C08959=1014.660,111.071,-128.777,-24.334,21.425,-41.690
C08960=1014.666,110.672,-128.741,-24.334,21.425,-41.694
C08961=1014.672,110.274,-128.704,-24.333,21.425,-41.697
C08962=1014.678,109.875,-128.668,-24.333,21.425,-41.701
C08963=1014.685,109.477,-128.631,-24.332,21.426,-41.703
C08964=1014.691,109.078,-128.595,-24.332,21.426,-41.707
C08965=1014.697,108.680,-128.557,-24.331,21.426,-41.710
C08966=1014.703,108.282,-128.521,-24.331,21.426,-41.714
C08967=1014.710,107.883,-128.485,-24.330,21.426,-41.717
C08968=1014.715,107.485,-128.448,-24.330,21.427,-41.719
C08969=1014.722,107.086,-128.411,-24.330,21.427,-41.723
C08970=1014.728,106.687,-128.374,-24.329,21.427,-41.727
C08971=1014.734,106.289,-128.338,-24.328,21.427,-41.730
C08972=1014.740,105.890,-128.301,-24.328,21.428,-41.734
C08973=1014.746,105.492,-128.265,-24.328,21.428,-41.736
C08974=1014.752,105.093,-128.228,-24.327,21.429,-41.740
C08975=1014.758,104.695,-128.192,-24.327,21.429,-41.743
C08976=1014.763,104.296,-128.155,-24.326,21.429,-41.747
C08977=1014.770,103.898,-128.118,-24.326,21.429,-41.751
C08978=1014.776,103.499,-128.082,-24.325,21.430,-41.754
C08979=1014.781,103.100,-128.044,-24.325,21.430,-41.756
C08980=1014.787,102.702,-128.008,-24.324,21.430,-41.760
C08981=1014.793,102.303,-127.972,-24.324,21.430,-41.763
C08982=1014.799,101.904,-127.935,-24.323,21.430,-41.767
C08983=1014.805,101.506,-127.898,-24.323,21.431,-41.771
C08984=1014.810,101.107,-127.862,-24.322,21.431,-41.775
C08985=1014.816,100.708,-127.826,-24.322,21.431,-41.778
C08986=1014.821,100.309,-127.789,-24.322,21.432,-41.780
C08987=1014.827,99.912,-127.752,-24.321,21.432,-41.784
C08988=1014.833,99.513,-127.716,-24.320,21.432,-41.787
C08989=1014.839,99.114,-127.679,-24.320,21.432,-41.791
C08990=1014.844,98.715,-127.643,-24.319,21.433,-41.795
C08991=1014.849,98.316,-127.606,-24.319,21.432,-41.798
C08992=1014.855,97.917,-127.569,-24.318,21.433,-41.802
C08993=1014.861,97.518,-127.533,-24.318,21.433,-41.806
C08994=1014.866,97.120,-127.497,-24.318,21.434,-41.808
C08995=1014.871,96.721,-127.459,-24.317,21.434,-41.811
C08996=1014.877,96.322,-127.423,-24.317,21.435,-41.815
C08997=1014.883,95.923,-127.386,-24.316,21.435,-41.819
C08998=1014.888,95.524,-127.350,-24.316,21.435,-41.822
C08999=1014.893,95.125,-127.314,-24.315,21.435,-41.826
C09000=1014.898,94.727,-127.277,-24.315,21.436,-41.830
C09001=1014.904,94.328,-127.240,-24.314,21.435,-41.833
C09002=1014.910,93.929,-127.204,-24.313,21.436,-41.837
C09003=1014.915,93.530,-127.168,-24.313,21.436,-41.841
C09004=1014.920,93.131,-127.131,-24.312,21.437,-41.844
C09005=1014.925,92.732,-127.095,-24.312,21.437,-41.846
C09006=1014.930,92.333,-127.057,-24.312,21.437,-41.850
C09007=1014.936,91.934,-127.021,-24.311,21.438,-41.854
C09008=1014.940,91.535,-126.985,-24.311,21.438,-41.857
C09009=1014.946,91.136,-126.948,-24.310,21.438,-41.861
C09010=1014.951,90.737,-126.912,-24.310,21.438,-41.865
C09011=1014.956,90.337,-126.875,-24.309,21.439,-41.868
C09012=1014.961,89.938,-126.839,-24.309,21.439,-41.872
C09013=1014.966,89.540,-126.802,-24.308,21.439,-41.875
C09014=1014.971,89.148,-126.766,-24.308,21.439,-41.879
C09015=1014.976,88.761,-126.731,-24.307,21.440,-41.883
C09016=1014.981,88.378,-126.696,-24.307,21.440,-41.887
C09017=1014.985,87.995,-126.662,-24.306,21.440,-41.890
C09018=1014.991,87.607,-126.625,-24.305,21.440,-41.894
C09019=1014.996,87.211,-126.590,-24.305,21.441,-41.898
C09020=1015.001,86.807,-126.553,-24.304,21.441,-41.901
C09021=1015.005,86.403,-126.516,-24.304,21.442,-41.905
C09022=1015.010,85.994,-126.479,-24.303,21.441,-41.908
C09023=1015.016,85.586,-126.441,-24.303,21.442,-41.912
C09024=1015.020,85.175,-126.405,-24.302,21.442,-41.916
C09025=1015.025,84.763,-126.366,-24.302,21.443,-41.920
C09026=1015.031,84.349,-126.328,-24.301,21.443,-41.923
C09027=1015.035,83.933,-126.291,-24.301,21.443,-41.927
C09028=1015.040,83.516,-126.253,-24.300,21.444,-41.931
C09029=1015.046,83.097,-126.214,-24.300,21.444,-41.935
C09030=1015.050,82.677,-126.176,-24.299,21.444,-41.938
C09031=1015.055,82.256,-126.138,-24.299,21.444,-41.942
C09032=1015.057,82.045,-126.118,-24.299,21.445,-41.944
C09033=1015.060,81.833,-126.099,-24.298,21.444,-41.947
C09034=1015.062,81.621,-126.080,-24.298,21.445,-41.949
C09035=1015.065,81.409,-126.061,-24.298,21.445,-41.951
C09036=1015.067,81.197,-126.041,-24.297,21.445,-41.953
C09037=1015.069,80.985,-126.022,-24.297,21.445,-41.955
C09038=1015.072,80.772,-126.002,-24.297,21.445,-41.956
C09039=1015.074,80.559,-125.983,-24.297,21.446,-41.958
C09040=1015.077,80.346,-125.963,-24.296,21.446,-41.960
C09041=1015.079,80.133,-125.945,-24.296,21.446,-41.962
C09042=1015.081,79.922,-125.925,-24.296,21.446,-41.964
C09043=1015.084,79.712,-125.906,-24.296,21.447,-41.966
C09044=1015.089,79.298,-125.869,-24.295,21.447,-41.970
C09045=1015.093,78.892,-125.831,-24.294,21.447,-41.973
C09046=1015.098,78.495,-125.795,-24.294,21.447,-41.977
C09047=1015.103,78.104,-125.760,-24.293,21.448,-41.980
C09048=1015.107,77.717,-125.725,-24.293,21.447,-41.986
C09049=1015.110,77.332,-125.690,-24.292,21.448,-41.989
C09050=1015.114,76.943,-125.655,-24.292,21.449,-41.994
C09051=1015.119,76.549,-125.619,-24.291,21.449,-41.997
C09052=1015.123,76.147,-125.582,-24.291,21.449,-42.001
C09053=1015.128,75.735,-125.545,-24.290,21.450,-42.004
C09054=1015.132,75.316,-125.507,-24.290,21.450,-42.008
C09055=1015.134,75.103,-125.487,-24.289,21.451,-42.010
C09056=1015.137,74.889,-125.468,-24.289,21.451,-42.012
C09057=1015.140,74.676,-125.449,-24.289,21.450,-42.015
C09058=1015.141,74.462,-125.430,-24.288,21.451,-42.017
C09059=1015.143,74.249,-125.409,-24.288,21.451,-42.019
C09060=1015.146,74.036,-125.391,-24.288,21.451,-42.021
C09061=1015.148,73.825,-125.372,-24.288,21.451,-42.023
C09062=1015.151,73.614,-125.352,-24.287,21.452,-42.025
C09063=1015.154,73.193,-125.314,-24.287,21.452,-42.028
C09064=1015.159,72.776,-125.276,-24.286,21.452,-42.034
C09065=1015.164,72.360,-125.239,-24.285,21.452,-42.037
C09066=1015.168,71.946,-125.201,-24.285,21.453,-42.041
C09067=1015.172,71.534,-125.164,-24.285,21.453,-42.045
C09068=1015.176,71.123,-125.127,-24.284,21.454,-42.049
C09069=1015.181,70.713,-125.090,-24.283,21.453,-42.054
C09070=1015.184,70.302,-125.052,-24.283,21.454,-42.058
C09071=1015.189,69.890,-125.015,-24.282,21.454,-42.061
C09072=1015.193,69.479,-124.978,-24.282,21.455,-42.065
C09073=1015.197,69.069,-124.941,-24.281,21.455,-42.069
C09074=1015.201,68.660,-124.904,-24.280,21.455,-42.074
C09075=1015.205,68.253,-124.867,-24.280,21.456,-42.078
C09076=1015.209,67.847,-124.830,-24.279,21.456,-42.082
C09077=1015.212,67.443,-124.794,-24.279,21.457,-42.085
C09078=1015.216,67.039,-124.757,-24.278,21.457,-42.089
C09079=1015.221,66.637,-124.721,-24.278,21.457,-42.094
C09080=1015.225,66.236,-124.685,-24.277,21.457,-42.098
C09081=1015.228,65.838,-124.649,-24.277,21.458,-42.102
C09082=1015.232,65.430,-124.612,-24.276,21.458,-42.106
C09083=1015.234,65.217,-124.593,-24.276,21.459,-42.108
C09084=1015.236,64.996,-124.574,-24.275,21.458,-42.111
C09085=1015.238,64.766,-124.553,-24.275,21.458,-42.113
C09086=1015.241,64.530,-124.531,-24.275,21.459,-42.115
C09087=1015.242,64.294,-124.510,-24.274,21.459,-42.116
C09088=1015.245,64.065,-124.489,-24.274,21.459,-42.120
C09089=1015.247,63.847,-124.470,-24.274,21.460,-42.122
C09090=1015.250,63.431,-124.432,-24.273,21.459,-42.127
C09091=1015.252,63.192,-124.410,-24.273,21.460,-42.129
C09092=1015.255,62.934,-124.387,-24.272,21.460,-42.131
C09093=1015.258,62.653,-124.362,-24.272,21.460,-42.133
C09094=1015.262,62.233,-124.324,-24.271,21.461,-42.139
C09095=1015.265,61.832,-124.289,-24.271,21.461,-42.142
C09096=1015.268,61.432,-124.252,-24.270,21.462,-42.146
C09097=1015.273,61.032,-124.217,-24.270,21.462,-42.150
C09098=1015.276,60.632,-124.181,-24.269,21.462,-42.155
C09099=1015.279,60.232,-124.145,-24.269,21.463,-42.159
C09100=1015.283,59.832,-124.109,-24.268,21.463,-42.163
C09101=1015.286,59.432,-124.072,-24.268,21.464,-42.166
C09102=1015.289,59.031,-124.037,-24.267,21.463,-42.172
C09103=1015.293,58.631,-124.000,-24.266,21.464,-42.175
C09104=1015.297,58.231,-123.965,-24.266,21.464,-42.179
C09105=1015.300,57.831,-123.929,-24.265,21.465,-42.183
C09106=1015.304,57.431,-123.894,-24.264,21.465,-42.188
C09107=1015.307,57.031,-123.858,-24.264,21.465,-42.192
C09108=1015.310,56.631,-123.822,-24.264,21.466,-42.196
C09109=1015.314,56.231,-123.785,-24.263,21.465,-42.201
C09110=1015.317,55.830,-123.750,-24.262,21.467,-42.205
C09111=1015.320,55.430,-123.714,-24.262,21.467,-42.209
C09112=1015.324,55.030,-123.679,-24.261,21.468,-42.212
C09113=1015.327,54.630,-123.642,-24.260,21.468,-42.218
C09114=1015.330,54.230,-123.607,-24.260,21.468,-42.221
C09115=1015.333,53.830,-123.571,-24.259,21.468,-42.225
C09116=1015.337,53.429,-123.536,-24.259,21.468,-42.230
C09117=1015.340,53.029,-123.499,-24.258,21.469,-42.234
C09118=1015.343,52.629,-123.464,-24.258,21.469,-42.238
C09119=1015.346,52.229,-123.428,-24.257,21.469,-42.243
C09120=1015.348,51.830,-123.392,-24.256,21.470,-42.247
C09121=1015.352,51.429,-123.357,-24.256,21.471,-42.251
C09122=1015.355,51.029,-123.321,-24.255,21.471,-42.255
C09123=1015.358,50.629,-123.285,-24.255,21.471,-42.260
C09124=1015.361,50.228,-123.249,-24.254,21.472,-42.264
C09125=1015.364,49.828,-123.214,-24.254,21.472,-42.268
C09126=1015.366,49.428,-123.178,-24.253,21.472,-42.273
C09127=1015.370,49.028,-123.143,-24.252,21.473,-42.277
C09128=1015.373,48.628,-123.106,-24.251,21.472,-42.282
C09129=1015.375,48.228,-123.072,-24.251,21.474,-42.286
C09130=1015.378,47.828,-123.036,-24.251,21.474,-42.290
C09131=1015.382,47.427,-123.000,-24.250,21.474,-42.295
C09132=1015.384,47.028,-122.965,-24.249,21.475,-42.299
C09133=1015.388,46.627,-122.929,-24.249,21.475,-42.302
C09134=1015.390,46.228,-122.894,-24.248,21.475,-42.308
C09135=1015.393,45.827,-122.858,-24.247,21.475,-42.311
C09136=1015.396,45.428,-122.823,-24.247,21.477,-42.316
C09137=1015.399,45.027,-122.787,-24.246,21.477,-42.321
C09138=1015.401,44.628,-122.752,-24.246,21.477,-42.325
C09139=1015.404,44.227,-122.716,-24.245,21.477,-42.330
C09140=1015.406,43.827,-122.681,-24.244,21.477,-42.333
C09141=1015.409,43.427,-122.646,-24.244,21.479,-42.338
C09142=1015.412,43.027,-122.610,-24.243,21.479,-42.343
C09143=1015.415,42.627,-122.575,-24.243,21.479,-42.347
C09144=1015.417,42.227,-122.539,-24.242,21.479,-42.352
C09145=1015.420,41.827,-122.504,-24.241,21.479,-42.356
C09146=1015.423,41.427,-122.468,-24.241,21.480,-42.359
C09147=1015.425,41.028,-122.433,-24.240,21.481,-42.365
C09148=1015.428,40.628,-122.398,-24.240,21.481,-42.369
C09149=1015.430,40.228,-122.362,-24.239,21.481,-42.374
C09150=1015.433,39.828,-122.327,-24.238,21.481,-42.378
C09151=1015.436,39.428,-122.292,-24.238,21.482,-42.383
C09152=1015.438,39.027,-122.256,-24.237,21.483,-42.387
C09153=1015.440,38.628,-122.221,-24.237,21.483,-42.391
C09154=1015.443,38.228,-122.186,-24.236,21.483,-42.396
C09155=1015.445,37.828,-122.151,-24.235,21.483,-42.400
C09156=1015.447,37.429,-122.115,-24.235,21.484,-42.405
C09157=1015.450,37.028,-122.080,-24.234,21.485,-42.409
C09158=1015.452,36.629,-122.045,-24.233,21.484,-42.414
C09159=1015.455,36.229,-122.010,-24.233,21.485,-42.418
C09160=1015.457,35.829,-121.974,-24.232,21.486,-42.424
C09161=1015.459,35.429,-121.940,-24.231,21.486,-42.428
C09162=1015.462,35.030,-121.905,-24.231,21.486,-42.433
C09163=1015.464,34.630,-121.869,-24.230,21.486,-42.437
C09164=1015.466,34.230,-121.834,-24.229,21.487,-42.442
C09165=1015.468,33.831,-121.799,-24.229,21.488,-42.446
C09166=1015.471,33.431,-121.764,-24.228,21.487,-42.451
C09167=1015.473,33.031,-121.729,-24.228,21.489,-42.455
C09168=1015.475,32.632,-121.694,-24.227,21.489,-42.461
C09169=1015.477,32.232,-121.659,-24.226,21.489,-42.464
C09170=1015.480,31.832,-121.624,-24.226,21.489,-42.469
C09171=1015.481,31.433,-121.589,-24.225,21.490,-42.474
C09172=1015.484,31.033,-121.554,-24.224,21.490,-42.479
C09173=1015.485,30.634,-121.519,-24.224,21.491,-42.483
C09174=1015.488,30.234,-121.484,-24.223,21.491,-42.488
C09175=1015.490,29.834,-121.449,-24.223,21.492,-42.492
C09176=1015.492,29.435,-121.414,-24.222,21.492,-42.497
C09177=1015.494,29.036,-121.379,-24.221,21.492,-42.501
C09178=1015.495,28.636,-121.345,-24.221,21.493,-42.507
C09179=1015.498,28.236,-121.309,-24.220,21.493,-42.510
C09180=1015.499,27.837,-121.274,-24.219,21.493,-42.516
C09181=1015.502,27.438,-121.240,-24.219,21.495,-42.520
C09182=1015.503,27.039,-121.205,-24.218,21.494,-42.525
C09183=1015.506,26.639,-121.170,-24.218,21.495,-42.529
C09184=1015.508,26.239,-121.136,-24.217,21.496,-42.534
C09185=1015.509,25.840,-121.101,-24.216,21.496,-42.540
C09186=1015.511,25.441,-121.066,-24.215,21.496,-42.543
C09187=1015.512,25.042,-121.031,-24.215,21.497,-42.549
C09188=1015.515,24.642,-120.997,-24.214,21.497,-42.553
C09189=1015.516,24.243,-120.962,-24.213,21.497,-42.558
C09190=1015.518,23.860,-120.929,-24.213,21.498,-42.562
C09191=1015.520,23.530,-120.899,-24.213,21.498,-42.564
C09192=1015.521,23.258,-120.876,-24.212,21.498,-42.567
C09193=1015.522,23.024,-120.856,-24.211,21.499,-42.573
C09194=1015.523,22.791,-120.836,-24.211,21.500,-42.577
C09195=1015.524,22.526,-120.812,-24.211,21.500,-42.580
C09196=1015.526,22.204,-120.785,-24.210,21.500,-42.584
C09197=1015.527,21.829,-120.752,-24.210,21.501,-42.586
C09198=1015.529,21.415,-120.717,-24.209,21.501,-42.593
C09199=1015.529,21.171,-120.695,-24.208,21.501,-42.597
C09200=1015.530,20.899,-120.671,-24.208,21.502,-42.599
C09201=1015.532,20.607,-120.647,-24.207,21.501,-42.602
C09202=1015.533,20.310,-120.621,-24.207,21.501,-42.604
C09203=1015.534,20.022,-120.596,-24.207,21.503,-42.606
C09204=1015.536,19.758,-120.573,-24.206,21.502,-42.610
C09205=1015.536,19.521,-120.552,-24.206,21.503,-42.613
C09206=1015.537,19.310,-120.535,-24.205,21.503,-42.617
C09207=1015.538,18.913,-120.500,-24.205,21.503,-42.622
C09208=1015.540,18.516,-120.466,-24.204,21.503,-42.626
C09209=1015.541,18.120,-120.431,-24.203,21.504,-42.632
C09210=1015.543,17.726,-120.398,-24.203,21.505,-42.635
C09211=1015.544,17.332,-120.363,-24.202,21.505,-42.641
C09212=1015.545,16.938,-120.330,-24.201,21.505,-42.646
C09213=1015.547,16.546,-120.296,-24.201,21.506,-42.650
C09214=1015.548,16.153,-120.262,-24.200,21.506,-42.656
C09215=1015.550,15.763,-120.228,-24.200,21.507,-42.659
C09216=1015.551,15.372,-120.195,-24.199,21.507,-42.665
C09217=1015.553,14.983,-120.161,-24.198,21.508,-42.670
C09218=1015.553,14.594,-120.128,-24.198,21.508,-42.674
C09219=1015.555,14.206,-120.094,-24.197,21.509,-42.680
C09220=1015.556,13.818,-120.061,-24.196,21.509,-42.683
C09221=1015.557,13.431,-120.028,-24.196,21.509,-42.689
C09222=1015.559,13.044,-119.994,-24.195,21.511,-42.693
C09223=1015.560,12.658,-119.961,-24.194,21.510,-42.698
C09224=1015.561,12.270,-119.929,-24.193,21.510,-42.703
C09225=1015.563,11.884,-119.895,-24.193,21.512,-42.707
C09226=1015.563,11.498,-119.862,-24.192,21.511,-42.713
C09227=1015.564,11.113,-119.829,-24.192,21.512,-42.716
C09228=1015.566,10.729,-119.796,-24.191,21.513,-42.722
C09229=1015.567,10.348,-119.764,-24.191,21.513,-42.726
C09230=1015.567,9.971,-119.732,-24.190,21.513,-42.731
C09231=1015.568,9.593,-119.699,-24.189,21.514,-42.737
C09232=1015.570,9.218,-119.667,-24.189,21.514,-42.740
C09233=1015.570,8.842,-119.635,-24.188,21.515,-42.746
C09234=1015.572,8.463,-119.602,-24.187,21.515,-42.751
C09235=1015.573,8.083,-119.570,-24.187,21.516,-42.755
C09236=1015.573,7.699,-119.537,-24.186,21.516,-42.761
C09237=1015.574,7.312,-119.504,-24.185,21.517,-42.764
C09238=1015.575,6.921,-119.471,-24.185,21.517,-42.770
C09239=1015.576,6.529,-119.437,-24.184,21.517,-42.775
C09240=1015.577,6.136,-119.404,-24.183,21.519,-42.779
C09241=1015.578,5.742,-119.371,-24.182,21.518,-42.785
C09242=1015.579,5.347,-119.337,-24.182,21.519,-42.790
C09243=1015.579,4.952,-119.304,-24.181,21.520,-42.794
C09244=1015.581,4.557,-119.270,-24.180,21.519,-42.799
C09245=1015.581,4.161,-119.237,-24.180,21.520,-42.805
C09246=1015.582,3.772,-119.203,-24.179,21.521,-42.809
C09247=1015.583,3.412,-119.172,-24.179,21.521,-42.812
C09248=1015.583,3.085,-119.145,-24.178,21.521,-42.817
C09249=1015.584,2.772,-119.119,-24.177,21.522,-42.823
C09250=1015.584,2.448,-119.091,-24.177,21.522,-42.827
C09251=1015.585,2.095,-119.061,-24.176,21.523,-42.833
C09252=1015.585,1.710,-119.028,-24.175,21.524,-42.836
C09253=1015.586,1.312,-118.995,-24.175,21.523,-42.841
C09254=1015.587,0.912,-118.961,-24.174,21.525,-42.846
C09255=1015.588,0.513,-118.928,-24.173,21.525,-42.851
C09256=1015.588,0.112,-118.893,-24.173,21.525,-42.857
C09257=1015.588,-0.292,-118.859,-24.172,21.525,-42.862
C09258=1015.590,-0.697,-118.826,-24.171,21.526,-42.867
C09259=1015.590,-1.105,-118.790,-24.171,21.527,-42.872
C09260=1015.591,-1.515,-118.756,-24.170,21.527,-42.877
C09261=1015.592,-1.928,-118.721,-24.169,21.528,-42.882
C09262=1015.592,-2.343,-118.687,-24.169,21.529,-42.888
C09263=1015.592,-2.760,-118.651,-24.168,21.529,-42.893
C09264=1015.593,-3.180,-118.615,-24.167,21.529,-42.899
C09265=1015.594,-3.601,-118.581,-24.166,21.530,-42.904
C09266=1015.594,-3.813,-118.563,-24.166,21.530,-42.908
C09267=1015.593,-4.025,-118.545,-24.165,21.530,-42.910
C09268=1015.594,-4.238,-118.527,-24.165,21.530,-42.913
C09269=1015.595,-4.454,-118.509,-24.165,21.531,-42.915
C09270=1015.594,-4.671,-118.491,-24.164,21.531,-42.919
C09271=1015.595,-4.889,-118.472,-24.164,21.531,-42.921
C09272=1015.595,-5.108,-118.453,-24.163,21.532,-42.925
C09273=1015.595,-5.330,-118.435,-24.163,21.532,-42.927
C09274=1015.595,-5.553,-118.417,-24.163,21.532,-42.930
C09275=1015.595,-5.776,-118.398,-24.162,21.532,-42.934
C09276=1015.595,-6.001,-118.379,-24.162,21.533,-42.935
C09277=1015.596,-6.224,-118.360,-24.161,21.533,-42.939
C09278=1015.595,-6.449,-118.341,-24.161,21.533,-42.941
C09279=1015.595,-6.673,-118.322,-24.161,21.533,-42.944
C09280=1015.596,-6.896,-118.304,-24.160,21.534,-42.947
C09281=1015.597,-7.119,-118.285,-24.160,21.534,-42.950
C09282=1015.597,-7.340,-118.266,-24.160,21.535,-42.952
C09283=1015.597,-7.560,-118.248,-24.159,21.534,-42.956
C09284=1015.596,-7.779,-118.230,-24.159,21.535,-42.959
C09285=1015.597,-7.998,-118.212,-24.158,21.535,-42.961
C09286=1015.597,-8.215,-118.193,-24.158,21.536,-42.965
C09287=1015.597,-8.432,-118.175,-24.158,21.536,-42.967
C09288=1015.597,-8.648,-118.157,-24.157,21.536,-42.971
C09289=1015.597,-8.864,-118.140,-24.157,21.537,-42.973
C09290=1015.598,-9.081,-118.121,-24.156,21.536,-42.976
C09291=1015.597,-9.298,-118.103,-24.156,21.537,-42.980
C09292=1015.598,-9.514,-118.085,-24.156,21.537,-42.982
C09293=1015.598,-9.731,-118.067,-24.155,21.538,-42.985
C09294=1015.598,-9.947,-118.049,-24.155,21.538,-42.987
C09295=1015.597,-10.163,-118.031,-24.154,21.538,-42.991
C09296=1015.598,-10.379,-118.013,-24.154,21.539,-42.993
C09297=1015.598,-10.593,-117.996,-24.154,21.538,-42.996
C09298=1015.598,-10.809,-117.977,-24.153,21.539,-42.998
C09299=1015.598,-11.023,-117.960,-24.153,21.539,-43.002
C09300=1015.598,-11.237,-117.941,-24.152,21.539,-43.006
C09301=1015.598,-11.451,-117.924,-24.152,21.540,-43.007
C09302=1015.598,-11.664,-117.906,-24.152,21.540,-43.011
C09303=1015.598,-11.877,-117.888,-24.151,21.540,-43.013
C09304=1015.598,-12.090,-117.871,-24.151,21.540,-43.016
C09305=1015.598,-12.301,-117.853,-24.151,21.541,-43.019
C09306=1015.598,-12.513,-117.835,-24.150,21.541,-43.022
C09307=1015.599,-12.724,-117.818,-24.150,21.542,-43.024
C09308=1015.598,-13.143,-117.783,-24.149,21.542,-43.029
C09309=1015.598,-13.561,-117.748,-24.148,21.543,-43.035
C09310=1015.598,-13.975,-117.715,-24.148,21.543,-43.041
C09311=1015.598,-14.387,-117.679,-24.147,21.544,-43.046
C09312=1015.598,-14.795,-117.645,-24.146,21.544,-43.052
C09313=1015.598,-15.201,-117.612,-24.145,21.545,-43.057
C09314=1015.597,-15.603,-117.579,-24.145,21.545,-43.063
C09315=1015.597,-16.004,-117.545,-24.144,21.546,-43.068
C09316=1015.597,-16.403,-117.513,-24.143,21.546,-43.074
C09317=1015.597,-16.803,-117.480,-24.142,21.547,-43.079
C09318=1015.597,-17.201,-117.447,-24.142,21.548,-43.085
C09319=1015.597,-17.598,-117.414,-24.141,21.547,-43.090
C09320=1015.596,-18.009,-117.380,-24.140,21.548,-43.098
C09321=1015.595,-18.258,-117.359,-24.139,21.549,-43.101
C09322=1015.595,-18.545,-117.336,-24.139,21.549,-43.105
C09323=1015.595,-18.856,-117.310,-24.139,21.550,-43.107
C09324=1015.595,-19.168,-117.285,-24.139,21.550,-43.109
C09325=1015.595,-19.455,-117.261,-24.138,21.550,-43.113
C09326=1015.595,-19.705,-117.240,-24.138,21.551,-43.116
C09327=1015.594,-20.116,-117.207,-24.136,21.551,-43.123
C09328=1015.593,-20.514,-117.174,-24.136,21.552,-43.129
C09329=1015.593,-20.912,-117.141,-24.135,21.553,-43.135
C09330=1015.592,-21.308,-117.108,-24.134,21.552,-43.140
C09331=1015.592,-21.706,-117.075,-24.134,21.553,-43.146
C09332=1015.591,-22.104,-117.043,-24.133,21.554,-43.151
C09333=1015.591,-22.501,-117.010,-24.132,21.554,-43.156
C09334=1015.590,-22.899,-116.978,-24.131,21.555,-43.162
C09335=1015.590,-23.296,-116.945,-24.131,21.555,-43.168
C09336=1015.589,-23.694,-116.913,-24.130,21.556,-43.173
C09337=1015.589,-24.092,-116.880,-24.129,21.556,-43.178
C09338=1015.588,-24.489,-116.848,-24.128,21.557,-43.184
C09339=1015.588,-24.886,-116.815,-24.128,21.558,-43.190
C09340=1015.587,-25.284,-116.782,-24.127,21.558,-43.195
C09341=1015.586,-25.682,-116.750,-24.126,21.558,-43.201
C09342=1015.585,-26.079,-116.718,-24.125,21.559,-43.206
C09343=1015.585,-26.476,-116.685,-24.125,21.560,-43.212
C09344=1015.584,-26.874,-116.653,-24.124,21.560,-43.217
C09345=1015.583,-27.272,-116.620,-24.123,21.561,-43.221
C09346=1015.582,-27.669,-116.588,-24.123,21.562,-43.227
C09347=1015.581,-28.066,-116.556,-24.122,21.562,-43.232
C09348=1015.581,-28.464,-116.523,-24.121,21.562,-43.238
C09349=1015.580,-28.862,-116.491,-24.120,21.563,-43.243
C09350=1015.579,-29.259,-116.459,-24.120,21.564,-43.249
C09351=1015.578,-29.656,-116.426,-24.119,21.565,-43.255
C09352=1015.577,-30.054,-116.394,-24.118,21.565,-43.260
C09353=1015.576,-30.451,-116.362,-24.117,21.565,-43.265
C09354=1015.575,-30.848,-116.329,-24.117,21.566,-43.271
C09355=1015.574,-31.246,-116.297,-24.116,21.567,-43.277
C09356=1015.573,-31.643,-116.265,-24.115,21.568,-43.282
C09357=1015.572,-32.041,-116.233,-24.114,21.567,-43.287
C09358=1015.571,-32.438,-116.201,-24.114,21.568,-43.293
C09359=1015.570,-32.836,-116.168,-24.113,21.569,-43.299
C09360=1015.569,-33.233,-116.136,-24.112,21.570,-43.304
C09361=1015.567,-33.630,-116.105,-24.111,21.570,-43.310
C09362=1015.566,-34.028,-116.072,-24.111,21.570,-43.315
C09363=1015.565,-34.425,-116.040,-24.110,21.571,-43.321
C09364=1015.564,-34.822,-116.008,-24.109,21.571,-43.328
C09365=1015.562,-35.220,-115.976,-24.108,21.572,-43.334
C09366=1015.562,-35.617,-115.944,-24.107,21.572,-43.339
C09367=1015.560,-36.014,-115.912,-24.107,21.573,-43.344
C09368=1015.559,-36.412,-115.879,-24.106,21.573,-43.350
C09369=1015.557,-36.809,-115.848,-24.105,21.574,-43.356
C09370=1015.557,-37.207,-115.816,-24.105,21.575,-43.361
C09371=1015.555,-37.605,-115.784,-24.104,21.575,-43.366
C09372=1015.554,-38.002,-115.752,-24.103,21.576,-43.372
C09373=1015.552,-38.399,-115.721,-24.102,21.576,-43.378
C09374=1015.551,-38.797,-115.688,-24.102,21.577,-43.383
C09375=1015.549,-39.194,-115.656,-24.101,21.578,-43.389
C09376=1015.547,-39.591,-115.625,-24.100,21.578,-43.394
C09377=1015.546,-39.988,-115.593,-24.099,21.579,-43.400
C09378=1015.545,-40.385,-115.561,-24.099,21.579,-43.405
C09379=1015.543,-40.783,-115.529,-24.098,21.580,-43.411
C09380=1015.541,-41.180,-115.497,-24.097,21.581,-43.417
C09381=1015.540,-41.577,-115.466,-24.096,21.582,-43.422
C09382=1015.538,-41.975,-115.434,-24.096,21.582,-43.427
C09383=1015.536,-42.371,-115.402,-24.095,21.582,-43.433
C09384=1015.535,-42.770,-115.370,-24.094,21.583,-43.439
C09385=1015.534,-43.167,-115.339,-24.093,21.584,-43.444
C09386=1015.532,-43.564,-115.307,-24.092,21.584,-43.451
C09387=1015.530,-43.962,-115.275,-24.092,21.585,-43.457
C09388=1015.528,-44.358,-115.244,-24.091,21.585,-43.462
C09389=1015.526,-44.756,-115.212,-24.090,21.585,-43.468
C09390=1015.524,-45.153,-115.181,-24.089,21.586,-43.473
C09391=1015.523,-45.550,-115.149,-24.089,21.587,-43.479
C09392=1015.521,-45.947,-115.117,-24.088,21.588,-43.485
C09393=1015.519,-46.344,-115.085,-24.087,21.589,-43.490
C09394=1015.518,-46.741,-115.054,-24.086,21.588,-43.496
C09395=1015.515,-47.138,-115.022,-24.086,21.589,-43.501
C09396=1015.513,-47.535,-114.991,-24.085,21.590,-43.507
C09397=1015.511,-47.934,-114.960,-24.084,21.591,-43.512
C09398=1015.509,-48.330,-114.929,-24.084,21.592,-43.518
C09399=1015.507,-48.728,-114.897,-24.083,21.592,-43.525
C09400=1015.505,-49.125,-114.866,-24.082,21.592,-43.531
C09401=1015.503,-49.521,-114.834,-24.081,21.592,-43.536
C09402=1015.501,-49.919,-114.803,-24.080,21.593,-43.542
C09403=1015.499,-50.316,-114.771,-24.080,21.594,-43.547
C09404=1015.496,-50.713,-114.740,-24.079,21.595,-43.553
C09405=1015.495,-51.110,-114.708,-24.078,21.595,-43.558
C09406=1015.492,-51.507,-114.677,-24.077,21.596,-43.564
C09407=1015.490,-51.904,-114.646,-24.077,21.597,-43.570
C09408=1015.488,-52.301,-114.614,-24.076,21.598,-43.575
C09409=1015.486,-52.697,-114.583,-24.075,21.598,-43.581
C09410=1015.483,-53.095,-114.552,-24.074,21.598,-43.588
C09411=1015.481,-53.491,-114.521,-24.073,21.599,-43.593
C09412=1015.478,-53.888,-114.490,-24.073,21.599,-43.599
C09413=1015.476,-54.286,-114.458,-24.072,21.600,-43.604
C09414=1015.474,-54.682,-114.427,-24.071,21.601,-43.610
C09415=1015.471,-55.079,-114.396,-24.071,21.602,-43.616
C09416=1015.469,-55.476,-114.365,-24.070,21.603,-43.621
C09417=1015.466,-55.874,-114.334,-24.069,21.602,-43.627
C09418=1015.464,-56.271,-114.303,-24.068,21.603,-43.632
C09419=1015.461,-56.669,-114.271,-24.067,21.603,-43.639
C09420=1015.459,-57.067,-114.240,-24.067,21.604,-43.645
C09421=1015.456,-57.466,-114.209,-24.066,21.605,-43.651
C09422=1015.453,-57.865,-114.177,-24.065,21.606,-43.656
C09423=1015.451,-58.264,-114.147,-24.064,21.606,-43.662
C09424=1015.448,-58.663,-114.115,-24.064,21.607,-43.667
C09425=1015.445,-59.063,-114.084,-24.063,21.608,-43.673
C09426=1015.442,-59.551,-114.046,-24.062,21.608,-43.680
C09427=1015.441,-59.865,-114.021,-24.061,21.609,-43.686
C09428=1015.437,-60.268,-113.990,-24.061,21.610,-43.691
C09429=1015.435,-60.670,-113.959,-24.060,21.610,-43.697
C09430=1015.432,-61.073,-113.928,-24.059,21.610,-43.702
C09431=1015.428,-61.476,-113.896,-24.058,21.611,-43.708
C09432=1015.426,-61.881,-113.864,-24.057,21.611,-43.715
C09433=1015.423,-62.285,-113.833,-24.057,21.612,-43.720
C09434=1015.419,-62.691,-113.802,-24.056,21.613,-43.726
C09435=1015.417,-63.096,-113.770,-24.055,21.614,-43.732
C09436=1015.413,-63.503,-113.738,-24.054,21.615,-43.737
C09437=1015.410,-63.910,-113.706,-24.053,21.615,-43.744
C09438=1015.407,-64.317,-113.675,-24.053,21.615,-43.750
C09439=1015.404,-64.724,-113.643,-24.052,21.616,-43.756
C09440=1015.401,-65.133,-113.612,-24.051,21.617,-43.761
C09441=1015.398,-65.541,-113.581,-24.050,21.617,-43.768
C09442=1015.394,-65.950,-113.548,-24.049,21.618,-43.774
C09443=1015.391,-66.360,-113.517,-24.049,21.619,-43.780
C09444=1015.388,-66.769,-113.485,-24.048,21.620,-43.785
C09445=1015.384,-67.178,-113.454,-24.047,21.620,-43.791
C09446=1015.381,-67.588,-113.422,-24.046,21.621,-43.798
C09447=1015.378,-67.999,-113.391,-24.046,21.621,-43.804
C09448=1015.374,-68.409,-113.358,-24.045,21.622,-43.809
C09449=1015.371,-68.820,-113.326,-24.044,21.623,-43.815
C09450=1015.367,-69.231,-113.295,-24.043,21.623,-43.822
C09451=1015.364,-69.641,-113.263,-24.042,21.624,-43.827
C09452=1015.360,-70.052,-113.231,-24.042,21.625,-43.833
C09453=1015.356,-70.463,-113.200,-24.041,21.625,-43.839
C09454=1015.353,-70.874,-113.169,-24.040,21.626,-43.846
C09455=1015.349,-71.285,-113.137,-24.039,21.626,-43.851
C09456=1015.345,-71.697,-113.105,-24.039,21.627,-43.857
C09457=1015.342,-72.107,-113.074,-24.038,21.628,-43.865
C09458=1015.338,-72.518,-113.042,-24.037,21.629,-43.870
C09459=1015.333,-72.929,-113.010,-24.036,21.630,-43.876
C09460=1015.330,-73.340,-112.979,-24.035,21.631,-43.881
C09461=1015.326,-73.750,-112.948,-24.034,21.631,-43.888
C09462=1015.322,-74.161,-112.916,-24.034,21.632,-43.894
C09463=1015.318,-74.571,-112.885,-24.033,21.632,-43.900
C09464=1015.315,-74.982,-112.853,-24.032,21.633,-43.905
C09465=1015.310,-75.392,-112.821,-24.031,21.633,-43.912
C09466=1015.306,-75.802,-112.790,-24.031,21.634,-43.918
C09467=1015.302,-76.211,-112.759,-24.030,21.635,-43.924
C09468=1015.298,-76.622,-112.728,-24.029,21.636,-43.929
C09469=1015.294,-77.031,-112.696,-24.028,21.636,-43.936
C09470=1015.290,-77.440,-112.666,-24.027,21.637,-43.942
C09471=1015.286,-77.847,-112.634,-24.027,21.637,-43.948
C09472=1015.282,-78.256,-112.603,-24.026,21.638,-43.953
C09473=1015.277,-78.664,-112.572,-24.025,21.638,-43.960
C09474=1015.274,-79.070,-112.541,-24.024,21.639,-43.966
C09475=1015.268,-79.477,-112.510,-24.023,21.640,-43.972
C09476=1015.264,-79.883,-112.479,-24.023,21.641,-43.977
C09477=1015.260,-80.289,-112.448,-24.022,21.641,-43.984
C09478=1015.256,-80.694,-112.417,-24.021,21.642,-43.990
C09479=1015.251,-81.099,-112.386,-24.020,21.643,-43.995
C09480=1015.247,-81.503,-112.356,-24.020,21.643,-44.001
C09481=1015.243,-81.906,-112.325,-24.019,21.644,-44.007
C09482=1015.238,-82.309,-112.294,-24.018,21.644,-44.014
C09483=1015.234,-82.711,-112.264,-24.017,21.645,-44.019
C09484=1015.229,-83.113,-112.234,-24.016,21.646,-44.025
C09485=1015.225,-83.514,-112.202,-24.016,21.647,-44.031
C09486=1015.220,-83.914,-112.172,-24.015,21.648,-44.036
C09487=1015.215,-84.313,-112.143,-24.014,21.648,-44.043
C09488=1015.211,-84.721,-112.111,-24.013,21.649,-44.049
C09489=1015.207,-84.944,-112.095,-24.013,21.649,-44.053
C09490=1015.204,-85.185,-112.076,-24.012,21.650,-44.056
C09491=1015.201,-85.438,-112.057,-24.012,21.649,-44.060
C09492=1015.199,-85.693,-112.038,-24.012,21.650,-44.062
C09493=1015.196,-85.939,-112.019,-24.011,21.650,-44.065
C09494=1015.194,-86.169,-112.002,-24.011,21.651,-44.069
C09495=1015.188,-86.578,-111.971,-24.010,21.652,-44.077
C09496=1015.183,-86.966,-111.941,-24.009,21.652,-44.082
C09497=1015.179,-87.346,-111.912,-24.008,21.652,-44.087
C09498=1015.174,-87.719,-111.884,-24.007,21.653,-44.093
C09499=1015.169,-88.090,-111.856,-24.007,21.654,-44.099
C09500=1015.164,-88.466,-111.828,-24.006,21.655,-44.104
C09501=1015.160,-88.873,-111.797,-24.005,21.656,-44.112
C09502=1015.157,-89.121,-111.778,-24.005,21.656,-44.116
C09503=1015.153,-89.396,-111.758,-24.004,21.657,-44.117
C09504=1015.150,-89.680,-111.737,-24.004,21.656,-44.121
C09505=1015.146,-89.954,-111.716,-24.003,21.657,-44.124
C09506=1015.143,-90.205,-111.697,-24.003,21.657,-44.128
C09507=1015.140,-90.423,-111.680,-24.002,21.658,-44.132
C09508=1015.135,-90.820,-111.651,-24.002,21.659,-44.138
C09509=1015.130,-91.213,-111.621,-24.001,21.659,-44.145
C09510=1015.125,-91.606,-111.591,-24.000,21.660,-44.150
C09511=1015.119,-91.998,-111.562,-23.999,21.660,-44.156
C09512=1015.114,-92.390,-111.532,-23.999,21.661,-44.162
C09513=1015.109,-92.781,-111.503,-23.998,21.662,-44.167
C09514=1015.103,-93.170,-111.474,-23.997,21.663,-44.173
C09515=1015.099,-93.560,-111.444,-23.996,21.664,-44.178
C09516=1015.093,-93.948,-111.415,-23.996,21.664,-44.184
C09517=1015.088,-94.336,-111.386,-23.995,21.664,-44.189
C09518=1015.083,-94.723,-111.357,-23.994,21.665,-44.195
C09519=1015.077,-95.109,-111.328,-23.994,21.666,-44.200
C09520=1015.071,-95.495,-111.299,-23.993,21.666,-44.207
C09521=1015.066,-95.880,-111.270,-23.992,21.667,-44.213
C09522=1015.061,-96.265,-111.241,-23.991,21.668,-44.219
C09523=1015.056,-96.649,-111.213,-23.990,21.668,-44.224
C09524=1015.049,-97.033,-111.183,-23.990,21.669,-44.230
C09525=1015.044,-97.415,-111.155,-23.989,21.669,-44.235
C09526=1015.038,-97.799,-111.127,-23.988,21.670,-44.241
C09527=1015.033,-98.183,-111.097,-23.988,21.671,-44.246
C09528=1015.027,-98.566,-111.068,-23.987,21.672,-44.252
C09529=1015.021,-98.950,-111.040,-23.986,21.673,-44.258
C09530=1015.015,-99.333,-111.011,-23.985,21.673,-44.263
C09531=1015.010,-99.717,-110.983,-23.985,21.673,-44.268
C09532=1015.004,-100.101,-110.954,-23.984,21.674,-44.274
C09533=1014.998,-100.486,-110.925,-23.983,21.675,-44.280
C09534=1014.992,-100.870,-110.896,-23.982,21.676,-44.285
C09535=1014.986,-101.257,-110.868,-23.982,21.677,-44.291
C09536=1014.980,-101.643,-110.839,-23.981,21.676,-44.296
C09537=1014.974,-102.030,-110.809,-23.980,21.677,-44.302
C09538=1014.968,-102.418,-110.780,-23.980,21.678,-44.307
C09539=1014.961,-102.807,-110.751,-23.979,21.678,-44.314
C09540=1014.955,-103.196,-110.723,-23.978,21.679,-44.320
C09541=1014.949,-103.586,-110.693,-23.977,21.680,-44.326
C09542=1014.943,-103.976,-110.664,-23.976,21.681,-44.331
C09543=1014.937,-104.368,-110.635,-23.976,21.682,-44.337
C09544=1014.930,-104.760,-110.606,-23.975,21.681,-44.342
C09545=1014.923,-105.151,-110.577,-23.974,21.682,-44.348
C09546=1014.917,-105.544,-110.548,-23.974,21.683,-44.353
C09547=1014.910,-105.937,-110.519,-23.973,21.684,-44.359
C09548=1014.904,-106.330,-110.489,-23.972,21.685,-44.365
C09549=1014.898,-106.723,-110.460,-23.971,21.686,-44.370
C09550=1014.890,-107.116,-110.431,-23.971,21.686,-44.376
C09551=1014.883,-107.509,-110.401,-23.970,21.687,-44.383
C09552=1014.877,-107.902,-110.372,-23.969,21.687,-44.388
C09553=1014.870,-108.295,-110.342,-23.968,21.688,-44.394
C09554=1014.863,-108.688,-110.314,-23.968,21.688,-44.399
C09555=1014.857,-109.082,-110.284,-23.967,21.689,-44.405
C09556=1014.849,-109.475,-110.255,-23.966,21.690,-44.411
C09557=1014.842,-109.867,-110.226,-23.965,21.691,-44.416
C09558=1014.835,-110.260,-110.197,-23.965,21.691,-44.422
C09559=1014.829,-110.653,-110.168,-23.964,21.692,-44.427
C09560=1014.821,-111.046,-110.138,-23.963,21.693,-44.433
C09561=1014.814,-111.439,-110.108,-23.963,21.694,-44.439
C09562=1014.807,-111.832,-110.080,-23.962,21.694,-44.446
C09563=1014.799,-112.224,-110.050,-23.961,21.694,-44.451
C09564=1014.792,-112.617,-110.021,-23.960,21.695,-44.456
C09565=1014.785,-113.010,-109.992,-23.959,21.696,-44.462
C09566=1014.777,-113.403,-109.963,-23.959,21.696,-44.468
C09567=1014.770,-113.795,-109.933,-23.958,21.697,-44.473
C09568=1014.762,-114.188,-109.905,-23.957,21.698,-44.479
C09569=1014.755,-114.581,-109.876,-23.957,21.699,-44.485
C09570=1014.748,-114.973,-109.846,-23.956,21.700,-44.490
C09571=1014.739,-115.366,-109.817,-23.955,21.701,-44.496
C09572=1014.732,-115.758,-109.788,-23.954,21.700,-44.501
C09573=1014.724,-116.151,-109.758,-23.954,21.701,-44.507
C09574=1014.716,-116.543,-109.730,-23.953,21.702,-44.512
C09575=1014.709,-116.936,-109.700,-23.952,21.703,-44.518
C09576=1014.700,-117.328,-109.671,-23.952,21.704,-44.523
C09577=1014.692,-117.721,-109.642,-23.951,21.705,-44.529
C09578=1014.685,-118.113,-109.613,-23.950,21.705,-44.536
C09579=1014.677,-118.506,-109.584,-23.949,21.705,-44.541
C09580=1014.668,-118.898,-109.555,-23.948,21.706,-44.547
C09581=1014.661,-119.291,-109.525,-23.948,21.706,-44.553
C09582=1014.652,-119.683,-109.496,-23.947,21.707,-44.558
C09583=1014.644,-120.076,-109.468,-23.946,21.708,-44.564
C09584=1014.636,-120.468,-109.439,-23.946,21.709,-44.569
C09585=1014.628,-120.860,-109.409,-23.945,21.710,-44.575
C09586=1014.619,-121.252,-109.380,-23.944,21.710,-44.580
C09587=1014.611,-121.645,-109.351,-23.943,21.710,-44.586
C09588=1014.603,-122.037,-109.322,-23.943,21.711,-44.591
C09589=1014.594,-122.429,-109.293,-23.942,21.712,-44.597
C09590=1014.586,-122.822,-109.264,-23.941,21.713,-44.603
C09591=1014.577,-123.214,-109.235,-23.941,21.714,-44.608
C09592=1014.568,-123.606,-109.206,-23.940,21.715,-44.614
C09593=1014.559,-123.998,-109.177,-23.939,21.714,-44.619
C09594=1014.551,-124.391,-109.148,-23.939,21.715,-44.625
C09595=1014.542,-124.782,-109.119,-23.938,21.716,-44.630
C09596=1014.533,-125.175,-109.090,-23.937,21.717,-44.636
C09597=1014.523,-125.567,-109.060,-23.936,21.718,-44.642
C09598=1014.515,-125.960,-109.031,-23.936,21.719,-44.647
C09599=1014.506,-126.351,-109.002,-23.935,21.719,-44.652
C09600=1014.497,-126.743,-108.972,-23.934,21.719,-44.658
C09601=1014.487,-127.136,-108.944,-23.934,21.720,-44.664
C09602=1014.478,-127.528,-108.914,-23.933,21.721,-44.669
C09603=1014.470,-127.920,-108.885,-23.932,21.722,-44.675
C09604=1014.460,-128.312,-108.856,-23.932,21.723,-44.680
C09605=1014.450,-128.704,-108.827,-23.931,21.723,-44.686
C09606=1014.441,-129.096,-108.798,-23.930,21.723,-44.691
C09607=1014.431,-129.488,-108.769,-23.929,21.724,-44.697
C09608=1014.422,-129.880,-108.740,-23.929,21.725,-44.703
C09609=1014.412,-130.272,-108.711,-23.928,21.726,-44.708
C09610=1014.402,-130.664,-108.681,-23.927,21.727,-44.714
C09611=1014.392,-131.056,-108.652,-23.926,21.727,-44.719
C09612=1014.383,-131.448,-108.623,-23.926,21.728,-44.725
C09613=1014.373,-131.841,-108.594,-23.925,21.728,-44.730
C09614=1014.364,-132.232,-108.565,-23.924,21.729,-44.736
C09615=1014.354,-132.625,-108.536,-23.924,21.730,-44.741
C09616=1014.343,-133.017,-108.507,-23.923,21.730,-44.747
C09617=1014.333,-133.409,-108.477,-23.922,21.731,-44.752
C09618=1014.324,-133.800,-108.448,-23.922,21.732,-44.758
C09619=1014.313,-134.192,-108.419,-23.921,21.732,-44.763
C09620=1014.765,-134.160,-108.701,-23.921,21.732,-44.763
C09621=1014.774,-133.768,-108.729,-23.922,21.732,-44.758
C09622=1014.784,-133.376,-108.758,-23.922,21.731,-44.752
C09623=1014.793,-132.984,-108.786,-23.923,21.730,-44.747
C09624=1014.802,-132.593,-108.815,-23.924,21.730,-44.741
C09625=1014.812,-132.200,-108.844,-23.924,21.729,-44.736
C09626=1014.821,-131.808,-108.872,-23.925,21.728,-44.730
C09627=1014.830,-131.417,-108.901,-23.926,21.728,-44.725
C09628=1014.838,-131.024,-108.930,-23.926,21.727,-44.719
C09629=1014.847,-130.632,-108.959,-23.927,21.727,-44.714
C09630=1014.857,-130.240,-108.988,-23.928,21.726,-44.708
C09631=1014.866,-129.848,-109.016,-23.929,21.725,-44.703
C09632=1014.874,-129.456,-109.045,-23.929,21.724,-44.697
C09633=1014.884,-129.064,-109.074,-23.930,21.723,-44.691
C09634=1014.892,-128.673,-109.102,-23.931,21.723,-44.686
C09635=1014.900,-128.280,-109.131,-23.932,21.723,-44.680
C09636=1014.909,-127.888,-109.159,-23.932,21.722,-44.675
C09637=1014.918,-127.495,-109.188,-23.933,21.721,-44.669
C09638=1014.927,-127.104,-109.217,-23.934,21.720,-44.664
C09639=1014.935,-126.712,-109.246,-23.934,21.719,-44.658
C09640=1014.943,-126.319,-109.275,-23.935,21.719,-44.652
C09641=1014.952,-125.928,-109.303,-23.936,21.719,-44.647
C09642=1014.960,-125.535,-109.332,-23.936,21.718,-44.642
C09643=1014.968,-125.143,-109.361,-23.937,21.717,-44.636
C09644=1014.977,-124.751,-109.389,-23.938,21.716,-44.630
C09645=1014.985,-124.359,-109.418,-23.939,21.715,-44.625
C09646=1014.993,-123.967,-109.447,-23.939,21.714,-44.619
C09647=1015.001,-123.575,-109.476,-23.940,21.715,-44.614
C09648=1015.009,-123.183,-109.504,-23.941,21.714,-44.608
C09649=1015.018,-122.790,-109.533,-23.941,21.713,-44.603
C09650=1015.025,-122.398,-109.562,-23.942,21.712,-44.597
C09651=1015.034,-122.006,-109.591,-23.943,21.711,-44.591
C09652=1015.041,-121.614,-109.619,-23.943,21.710,-44.586
C09653=1015.050,-121.222,-109.648,-23.944,21.710,-44.580
C09654=1015.056,-120.829,-109.677,-23.945,21.710,-44.575
C09655=1015.064,-120.437,-109.705,-23.946,21.709,-44.569
C09656=1015.072,-120.045,-109.734,-23.946,21.708,-44.564
C09657=1015.080,-119.652,-109.764,-23.947,21.707,-44.558
C09658=1015.088,-119.259,-109.792,-23.948,21.706,-44.553
C09659=1015.095,-118.867,-109.821,-23.948,21.706,-44.547
C09660=1015.102,-118.475,-109.850,-23.949,21.705,-44.541
C09661=1015.111,-118.083,-109.879,-23.950,21.705,-44.536
C09662=1015.117,-117.690,-109.907,-23.951,21.705,-44.529
C09663=1015.125,-117.298,-109.936,-23.952,21.704,-44.523
C09664=1015.132,-116.905,-109.965,-23.952,21.703,-44.518
C09665=1015.139,-116.513,-109.994,-23.953,21.702,-44.512
C09666=1015.147,-116.121,-110.022,-23.954,21.701,-44.507
C09667=1015.154,-115.728,-110.051,-23.954,21.700,-44.501
C09668=1015.161,-115.335,-110.081,-23.955,21.701,-44.496
C09669=1015.168,-114.943,-110.109,-23.956,21.700,-44.490
C09670=1015.175,-114.550,-110.138,-23.957,21.699,-44.485
C09671=1015.183,-114.158,-110.166,-23.957,21.698,-44.479
C09672=1015.190,-113.765,-110.196,-23.958,21.697,-44.473
C09673=1015.197,-113.372,-110.224,-23.959,21.696,-44.468
C09674=1015.204,-112.980,-110.253,-23.959,21.696,-44.462
C09675=1015.210,-112.587,-110.282,-23.960,21.695,-44.456
C09676=1015.217,-112.194,-110.311,-23.961,21.694,-44.451
C09677=1015.224,-111.802,-110.341,-23.962,21.694,-44.446
C09678=1015.231,-111.409,-110.369,-23.963,21.694,-44.439
C09679=1015.238,-111.016,-110.397,-23.963,21.693,-44.433
C09680=1015.244,-110.622,-110.427,-23.964,21.692,-44.427
C09681=1015.251,-110.230,-110.456,-23.965,21.691,-44.422
C09682=1015.258,-109.837,-110.485,-23.965,21.691,-44.416
C09683=1015.264,-109.444,-110.514,-23.966,21.690,-44.411
C09684=1015.271,-109.051,-110.543,-23.967,21.689,-44.405
C09685=1015.277,-108.658,-110.572,-23.968,21.688,-44.399
C09686=1015.284,-108.265,-110.600,-23.968,21.688,-44.394
C09687=1015.290,-107.873,-110.630,-23.969,21.687,-44.388
C09688=1015.297,-107.479,-110.659,-23.970,21.687,-44.383
C09689=1015.303,-107.086,-110.688,-23.971,21.686,-44.376
C09690=1015.309,-106.693,-110.717,-23.971,21.686,-44.370
C09691=1015.315,-106.300,-110.746,-23.972,21.685,-44.365
C09692=1015.322,-105.907,-110.775,-23.973,21.684,-44.359
C09693=1015.328,-105.514,-110.804,-23.974,21.683,-44.353
C09694=1015.334,-105.122,-110.833,-23.974,21.682,-44.348
C09695=1015.340,-104.730,-110.862,-23.975,21.681,-44.342
C09696=1015.346,-104.338,-110.891,-23.976,21.682,-44.337
C09697=1015.352,-103.947,-110.920,-23.976,21.681,-44.331
C09698=1015.358,-103.557,-110.949,-23.977,21.680,-44.326
C09699=1015.364,-103.167,-110.978,-23.978,21.679,-44.320
C09700=1015.370,-102.777,-111.007,-23.979,21.678,-44.314
C09701=1015.376,-102.389,-111.035,-23.980,21.678,-44.307
C09702=1015.382,-102.001,-111.063,-23.980,21.677,-44.302
C09703=1015.387,-101.614,-111.093,-23.981,21.676,-44.296
C09704=1015.393,-101.227,-111.121,-23.982,21.677,-44.291
C09705=1015.399,-100.842,-111.150,-23.982,21.676,-44.285
C09706=1015.405,-100.457,-111.178,-23.983,21.675,-44.280
C09707=1015.410,-100.072,-111.207,-23.984,21.674,-44.274
C09708=1015.415,-99.688,-111.236,-23.985,21.673,-44.268
C09709=1015.421,-99.304,-111.264,-23.985,21.673,-44.263
C09710=1015.427,-98.920,-111.293,-23.986,21.673,-44.258
C09711=1015.432,-98.537,-111.321,-23.987,21.672,-44.252
C09712=1015.438,-98.154,-111.350,-23.988,21.671,-44.246
C09713=1015.442,-97.802,-111.376,-23.988,21.670,-44.241
C09714=1015.448,-97.387,-111.407,-23.989,21.669,-44.235
C09715=1015.453,-97.003,-111.436,-23.990,21.669,-44.230
C09716=1015.458,-96.619,-111.464,-23.990,21.668,-44.224
C09717=1015.464,-96.235,-111.492,-23.991,21.668,-44.219
C09718=1015.469,-95.850,-111.521,-23.992,21.667,-44.213
C09719=1015.474,-95.466,-111.550,-23.993,21.666,-44.207
C09720=1015.479,-95.080,-111.579,-23.994,21.666,-44.200
C09721=1015.484,-94.694,-111.608,-23.994,21.665,-44.195
C09722=1015.489,-94.307,-111.637,-23.995,21.664,-44.189
C09723=1015.494,-93.919,-111.666,-23.996,21.664,-44.184
C09724=1015.500,-93.531,-111.695,-23.996,21.664,-44.178
C09725=1015.504,-93.142,-111.723,-23.997,21.663,-44.173
C09726=1015.510,-92.751,-111.752,-23.998,21.662,-44.167
C09727=1015.514,-92.361,-111.782,-23.999,21.661,-44.162
C09728=1015.520,-91.969,-111.811,-23.999,21.660,-44.156
C09729=1015.525,-91.577,-111.841,-24.000,21.660,-44.150
C09730=1015.529,-91.184,-111.870,-24.001,21.659,-44.145
C09731=1015.534,-90.791,-111.900,-24.002,21.659,-44.138
C09732=1015.540,-90.395,-111.929,-24.002,21.658,-44.132
C09733=1015.542,-90.176,-111.945,-24.003,21.657,-44.128
C09734=1015.545,-89.926,-111.964,-24.003,21.657,-44.124
C09735=1015.548,-89.651,-111.985,-24.004,21.656,-44.121
C09736=1015.551,-89.367,-112.007,-24.004,21.657,-44.117
C09737=1015.555,-89.092,-112.027,-24.005,21.656,-44.116
C09738=1015.558,-88.844,-112.045,-24.005,21.656,-44.112
C09739=1015.563,-88.437,-112.076,-24.006,21.655,-44.104
C09740=1015.567,-88.062,-112.104,-24.007,21.654,-44.099
C09741=1015.571,-87.690,-112.132,-24.007,21.653,-44.093
C09742=1015.576,-87.317,-112.160,-24.008,21.652,-44.087
C09743=1015.580,-86.938,-112.189,-24.009,21.652,-44.082
C09744=1015.585,-86.550,-112.218,-24.010,21.652,-44.077
C09745=1015.590,-86.140,-112.248,-24.011,21.651,-44.069
C09746=1015.592,-85.911,-112.265,-24.011,21.650,-44.065
C09747=1015.595,-85.664,-112.284,-24.012,21.650,-44.062
C09748=1015.597,-85.410,-112.304,-24.012,21.649,-44.060
C09749=1015.600,-85.156,-112.322,-24.012,21.650,-44.056
C09750=1015.603,-84.915,-112.341,-24.013,21.649,-44.053
C09751=1015.605,-84.691,-112.358,-24.013,21.649,-44.049
C09752=1015.610,-84.285,-112.389,-24.014,21.648,-44.043
C09753=1015.614,-83.886,-112.419,-24.015,21.648,-44.036
C09754=1015.619,-83.485,-112.449,-24.016,21.647,-44.031
C09755=1015.624,-83.084,-112.479,-24.016,21.646,-44.025
C09756=1015.628,-82.682,-112.510,-24.017,21.645,-44.019
C09757=1015.632,-82.280,-112.540,-24.018,21.644,-44.014
C09758=1015.636,-81.877,-112.570,-24.019,21.644,-44.007
C09759=1015.640,-81.474,-112.601,-24.020,21.643,-44.001
C09760=1015.645,-81.070,-112.631,-24.020,21.643,-43.995
C09761=1015.649,-80.665,-112.662,-24.021,21.642,-43.990
C09762=1015.653,-80.260,-112.693,-24.022,21.641,-43.984
C09763=1015.657,-79.855,-112.723,-24.023,21.641,-43.977
C09764=1015.661,-79.449,-112.755,-24.023,21.640,-43.972
C09765=1015.666,-79.042,-112.786,-24.024,21.639,-43.966
C09766=1015.669,-78.635,-112.817,-24.025,21.638,-43.960
C09767=1015.673,-78.227,-112.847,-24.026,21.638,-43.953
C09768=1015.678,-77.820,-112.878,-24.027,21.637,-43.948
C09769=1015.681,-77.411,-112.910,-24.027,21.637,-43.942
C09770=1015.685,-77.002,-112.940,-24.028,21.636,-43.936
C09771=1015.689,-76.593,-112.972,-24.029,21.636,-43.929
C09772=1015.693,-76.184,-113.002,-24.030,21.635,-43.924
C09773=1015.697,-75.774,-113.034,-24.031,21.634,-43.918
C09774=1015.701,-75.364,-113.065,-24.031,21.633,-43.912
C09775=1015.704,-74.954,-113.097,-24.032,21.633,-43.905
C09776=1015.708,-74.543,-113.128,-24.033,21.632,-43.900
C09777=1015.713,-74.133,-113.159,-24.034,21.632,-43.894
C09778=1015.716,-73.722,-113.191,-24.034,21.631,-43.888
C09779=1015.720,-73.311,-113.222,-24.035,21.631,-43.881
C09780=1015.724,-72.901,-113.253,-24.036,21.630,-43.876
C09781=1015.727,-72.490,-113.285,-24.037,21.629,-43.870
C09782=1015.731,-72.079,-113.317,-24.038,21.628,-43.865
C09783=1015.734,-71.668,-113.348,-24.039,21.627,-43.857
C09784=1015.737,-71.257,-113.379,-24.039,21.626,-43.851
C09785=1015.742,-70.846,-113.411,-24.040,21.626,-43.846
C09786=1015.745,-70.436,-113.442,-24.041,21.625,-43.839
C09787=1015.748,-70.024,-113.473,-24.042,21.625,-43.833
C09788=1015.752,-69.613,-113.505,-24.042,21.624,-43.827
C09789=1015.755,-69.203,-113.537,-24.043,21.623,-43.822
C09790=1015.759,-68.792,-113.569,-24.044,21.623,-43.815
C09791=1015.762,-68.381,-113.600,-24.045,21.622,-43.809
C09792=1015.765,-67.971,-113.632,-24.046,21.621,-43.804
C09793=1015.768,-67.561,-113.663,-24.046,21.621,-43.798
C09794=1015.771,-67.151,-113.695,-24.047,21.620,-43.791
C09795=1015.775,-66.740,-113.727,-24.048,21.620,-43.785
C09796=1015.778,-66.332,-113.758,-24.049,21.619,-43.780
C09797=1015.781,-65.922,-113.789,-24.049,21.618,-43.774
C09798=1015.784,-65.513,-113.821,-24.050,21.617,-43.768
C09799=1015.788,-65.105,-113.853,-24.051,21.617,-43.761
C09800=1015.790,-64.696,-113.885,-24.052,21.616,-43.756
C09801=1015.793,-64.289,-113.916,-24.053,21.615,-43.750
C09802=1015.796,-63.882,-113.948,-24.053,21.615,-43.744
C09803=1015.799,-63.475,-113.979,-24.054,21.615,-43.737
C09804=1015.802,-63.068,-114.010,-24.055,21.614,-43.732
C09805=1015.805,-62.663,-114.042,-24.056,21.613,-43.726
C09806=1015.808,-62.257,-114.073,-24.057,21.612,-43.720
C09807=1015.811,-61.853,-114.104,-24.057,21.611,-43.715
C09808=1015.814,-61.449,-114.136,-24.058,21.611,-43.708
C09809=1015.817,-61.045,-114.167,-24.059,21.610,-43.702
C09810=1015.820,-60.643,-114.199,-24.060,21.610,-43.697
C09811=1015.822,-60.239,-114.230,-24.061,21.610,-43.691
C09812=1015.824,-59.837,-114.261,-24.061,21.609,-43.686
C09813=1015.827,-59.437,-114.293,-24.062,21.608,-43.680
C09814=1015.830,-59.035,-114.324,-24.063,21.608,-43.673
C09815=1015.833,-58.635,-114.355,-24.064,21.607,-43.667
C09816=1015.835,-58.236,-114.386,-24.064,21.606,-43.662
C09817=1015.837,-57.836,-114.417,-24.065,21.606,-43.656
C09818=1015.840,-57.438,-114.448,-24.066,21.605,-43.651
C09819=1015.842,-57.039,-114.480,-24.067,21.604,-43.645
C09820=1015.845,-56.642,-114.510,-24.067,21.603,-43.639
C09821=1015.847,-56.244,-114.542,-24.068,21.603,-43.632
C09822=1015.849,-55.846,-114.573,-24.069,21.602,-43.627
C09823=1015.852,-55.449,-114.604,-24.070,21.603,-43.621
C09824=1015.854,-55.052,-114.635,-24.071,21.602,-43.616
C09825=1015.857,-54.654,-114.666,-24.071,21.601,-43.610
C09826=1015.859,-54.257,-114.697,-24.072,21.600,-43.604
C09827=1015.861,-53.861,-114.728,-24.073,21.599,-43.599
C09828=1015.864,-53.463,-114.760,-24.073,21.599,-43.593
C09829=1015.866,-53.067,-114.791,-24.074,21.598,-43.588
C09830=1015.868,-52.670,-114.822,-24.075,21.598,-43.581
C09831=1015.870,-52.273,-114.853,-24.076,21.598,-43.575
C09832=1015.872,-51.876,-114.885,-24.077,21.597,-43.570
C09833=1015.875,-51.479,-114.916,-24.077,21.596,-43.564
C09834=1015.877,-51.082,-114.947,-24.078,21.595,-43.558
C09835=1015.878,-50.686,-114.978,-24.079,21.595,-43.553
C09836=1015.881,-50.288,-115.009,-24.080,21.594,-43.547
C09837=1015.882,-49.891,-115.041,-24.080,21.593,-43.542
C09838=1015.885,-49.494,-115.072,-24.081,21.592,-43.536
C09839=1015.887,-49.096,-115.104,-24.082,21.592,-43.531
C09840=1015.889,-48.700,-115.135,-24.083,21.592,-43.525
C09841=1015.891,-48.303,-115.166,-24.084,21.592,-43.518
C09842=1015.893,-47.905,-115.198,-24.084,21.591,-43.512
C09843=1015.895,-47.509,-115.229,-24.085,21.590,-43.507
C09844=1015.896,-47.111,-115.260,-24.086,21.589,-43.501
C09845=1015.898,-46.713,-115.292,-24.086,21.588,-43.496
C09846=1015.900,-46.317,-115.323,-24.087,21.589,-43.490
C09847=1015.902,-45.920,-115.354,-24.088,21.588,-43.485
C09848=1015.904,-45.522,-115.386,-24.089,21.587,-43.479
C09849=1015.906,-45.125,-115.418,-24.089,21.586,-43.473
C09850=1015.907,-44.728,-115.450,-24.090,21.585,-43.468
C09851=1015.909,-44.331,-115.482,-24.091,21.585,-43.462
C09852=1015.910,-43.933,-115.512,-24.092,21.585,-43.457
C09853=1015.912,-43.536,-115.544,-24.092,21.584,-43.451
C09854=1015.914,-43.139,-115.576,-24.093,21.584,-43.444
C09855=1015.916,-42.742,-115.608,-24.094,21.583,-43.439
C09856=1015.917,-42.345,-115.639,-24.095,21.582,-43.433
C09857=1015.919,-41.947,-115.671,-24.096,21.582,-43.427
C09858=1015.921,-41.550,-115.703,-24.096,21.582,-43.422
C09859=1015.921,-41.152,-115.734,-24.097,21.581,-43.417
C09860=1015.923,-40.755,-115.766,-24.098,21.580,-43.411
C09861=1015.925,-40.358,-115.798,-24.099,21.579,-43.405
C09862=1015.926,-39.961,-115.829,-24.099,21.579,-43.400
C09863=1015.927,-39.564,-115.861,-24.100,21.578,-43.394
C09864=1015.929,-39.166,-115.893,-24.101,21.578,-43.389
C09865=1015.931,-38.769,-115.925,-24.102,21.577,-43.383
C09866=1015.931,-38.372,-115.957,-24.102,21.576,-43.378
C09867=1015.934,-37.974,-115.989,-24.103,21.576,-43.372
C09868=1015.934,-37.576,-116.021,-24.104,21.575,-43.366
C09869=1015.936,-37.179,-116.052,-24.105,21.575,-43.361
C09870=1015.937,-36.781,-116.085,-24.105,21.574,-43.356
C09871=1015.938,-36.385,-116.116,-24.106,21.573,-43.350
C09872=1015.939,-35.987,-116.149,-24.107,21.573,-43.344
C09873=1015.941,-35.590,-116.180,-24.107,21.572,-43.339
C09874=1015.942,-35.192,-116.213,-24.108,21.572,-43.334
C09875=1015.943,-34.795,-116.245,-24.109,21.571,-43.328
C09876=1015.944,-34.398,-116.276,-24.110,21.571,-43.321
C09877=1015.946,-34.000,-116.309,-24.111,21.570,-43.315
C09878=1015.946,-33.602,-116.340,-24.111,21.570,-43.310
C09879=1015.948,-33.206,-116.372,-24.112,21.570,-43.304
C09880=1015.948,-32.808,-116.404,-24.113,21.569,-43.299
C09881=1015.950,-32.410,-116.437,-24.114,21.568,-43.293
C09882=1015.951,-32.013,-116.469,-24.114,21.567,-43.287
C09883=1015.951,-31.616,-116.501,-24.115,21.568,-43.282
C09884=1015.952,-31.219,-116.533,-24.116,21.567,-43.277
C09885=1015.953,-30.821,-116.566,-24.117,21.566,-43.271
C09886=1015.954,-30.423,-116.598,-24.117,21.565,-43.265
C09887=1015.955,-30.026,-116.630,-24.118,21.565,-43.260
C09888=1015.956,-29.629,-116.662,-24.119,21.565,-43.255
C09889=1015.957,-29.231,-116.695,-24.120,21.564,-43.249
C09890=1015.958,-28.834,-116.727,-24.120,21.563,-43.243
C09891=1015.959,-28.437,-116.759,-24.121,21.562,-43.238
C09892=1015.959,-28.039,-116.792,-24.122,21.562,-43.232
C09893=1015.961,-27.641,-116.824,-24.123,21.562,-43.227
C09894=1015.962,-27.244,-116.856,-24.123,21.561,-43.221
C09895=1015.962,-26.847,-116.888,-24.124,21.560,-43.217
C09896=1015.962,-26.449,-116.921,-24.125,21.560,-43.212
C09897=1015.963,-26.052,-116.953,-24.125,21.559,-43.206
C09898=1015.965,-25.654,-116.986,-24.126,21.558,-43.201
C09899=1015.965,-25.257,-117.019,-24.127,21.558,-43.195
C09900=1015.965,-24.859,-117.051,-24.128,21.558,-43.190
C09901=1015.966,-24.462,-117.083,-24.128,21.557,-43.184
C09902=1015.966,-24.064,-117.116,-24.129,21.556,-43.178
C09903=1015.968,-23.667,-117.148,-24.130,21.556,-43.173
C09904=1015.968,-23.269,-117.181,-24.131,21.555,-43.168
C09905=1015.968,-22.872,-117.213,-24.131,21.555,-43.162
C09906=1015.968,-22.474,-117.246,-24.132,21.554,-43.156
C09907=1015.969,-22.077,-117.278,-24.133,21.554,-43.151
C09908=1015.970,-21.679,-117.312,-24.134,21.553,-43.146
C09909=1015.971,-21.281,-117.344,-24.134,21.552,-43.140
C09910=1015.971,-20.884,-117.377,-24.135,21.553,-43.135
C09911=1015.971,-20.486,-117.409,-24.136,21.552,-43.129
C09912=1015.971,-20.089,-117.441,-24.136,21.551,-43.123
C09913=1015.972,-19.677,-117.476,-24.138,21.551,-43.116
C09914=1015.972,-19.428,-117.497,-24.138,21.550,-43.113
C09915=1015.972,-19.140,-117.520,-24.139,21.550,-43.109
C09916=1015.973,-18.829,-117.546,-24.139,21.550,-43.107
C09917=1015.973,-18.518,-117.571,-24.139,21.549,-43.105
C09918=1015.973,-18.230,-117.595,-24.139,21.549,-43.101
C09919=1015.974,-17.982,-117.615,-24.140,21.548,-43.098
C09920=1015.974,-17.571,-117.649,-24.141,21.547,-43.090
C09921=1015.974,-17.173,-117.682,-24.142,21.548,-43.085
C09922=1015.974,-16.776,-117.715,-24.142,21.547,-43.079
C09923=1015.974,-16.377,-117.748,-24.143,21.546,-43.074
C09924=1015.975,-15.977,-117.781,-24.144,21.546,-43.068
C09925=1015.974,-15.577,-117.814,-24.145,21.545,-43.063
C09926=1015.975,-15.173,-117.848,-24.145,21.545,-43.057
C09927=1015.975,-14.768,-117.881,-24.146,21.544,-43.052
C09928=1015.975,-14.360,-117.915,-24.147,21.544,-43.046
C09929=1015.975,-13.948,-117.949,-24.148,21.543,-43.041
C09930=1015.975,-13.533,-117.984,-24.148,21.543,-43.035
C09931=1015.975,-13.116,-118.018,-24.149,21.542,-43.029
C09932=1015.975,-12.697,-118.053,-24.150,21.542,-43.024
C09933=1015.975,-12.485,-118.070,-24.150,21.541,-43.022
C09934=1015.976,-12.274,-118.088,-24.151,21.541,-43.019
C09935=1015.975,-12.062,-118.106,-24.151,21.540,-43.016
C09936=1015.975,-11.850,-118.123,-24.151,21.540,-43.013
C09937=1015.975,-11.637,-118.141,-24.152,21.540,-43.011
C09938=1015.975,-11.424,-118.159,-24.152,21.540,-43.007
C09939=1015.975,-11.211,-118.177,-24.152,21.539,-43.006
C09940=1015.975,-10.996,-118.194,-24.153,21.539,-43.002
C09941=1015.975,-10.781,-118.213,-24.153,21.539,-42.998
C09942=1015.975,-10.567,-118.230,-24.154,21.538,-42.996
C09943=1015.975,-10.351,-118.248,-24.154,21.539,-42.993
C09944=1015.975,-10.135,-118.266,-24.154,21.538,-42.991
C09945=1015.975,-9.920,-118.284,-24.155,21.538,-42.987
C09946=1015.975,-9.703,-118.303,-24.155,21.538,-42.985
C09947=1015.974,-9.487,-118.320,-24.156,21.537,-42.982
C09948=1015.975,-9.270,-118.338,-24.156,21.537,-42.980
C09949=1015.974,-9.054,-118.356,-24.156,21.536,-42.976
C09950=1015.974,-8.838,-118.374,-24.157,21.537,-42.973
C09951=1015.974,-8.621,-118.393,-24.157,21.536,-42.971
C09952=1015.974,-8.404,-118.411,-24.158,21.536,-42.967
C09953=1015.974,-8.187,-118.429,-24.158,21.536,-42.965
C09954=1015.974,-7.970,-118.447,-24.158,21.535,-42.961
C09955=1015.974,-7.752,-118.465,-24.159,21.535,-42.959
C09956=1015.973,-7.533,-118.483,-24.159,21.534,-42.956
C09957=1015.974,-7.312,-118.502,-24.160,21.535,-42.952
C09958=1015.974,-7.092,-118.521,-24.160,21.534,-42.950
C09959=1015.973,-6.869,-118.539,-24.160,21.534,-42.947
C09960=1015.973,-6.645,-118.557,-24.161,21.533,-42.944
C09961=1015.973,-6.421,-118.576,-24.161,21.533,-42.941
C09962=1015.973,-6.198,-118.595,-24.161,21.533,-42.939
C09963=1015.973,-5.973,-118.615,-24.162,21.533,-42.935
C09964=1015.972,-5.749,-118.633,-24.162,21.532,-42.934
C09965=1015.972,-5.526,-118.652,-24.163,21.532,-42.930
C09966=1015.972,-5.303,-118.670,-24.163,21.532,-42.927
C09967=1015.972,-5.081,-118.688,-24.163,21.532,-42.925
C09968=1015.972,-4.861,-118.708,-24.164,21.531,-42.921
C09969=1015.972,-4.643,-118.726,-24.164,21.531,-42.919
C09970=1015.971,-4.427,-118.744,-24.165,21.531,-42.915
C09971=1015.971,-4.211,-118.762,-24.165,21.530,-42.913
C09972=1015.971,-3.997,-118.780,-24.165,21.530,-42.910
C09973=1015.971,-3.786,-118.798,-24.166,21.530,-42.908
C09974=1015.970,-3.573,-118.815,-24.166,21.530,-42.904
C09975=1015.970,-3.152,-118.851,-24.167,21.529,-42.899
C09976=1015.969,-2.733,-118.886,-24.168,21.529,-42.893
C09977=1015.969,-2.316,-118.922,-24.169,21.529,-42.888
C09978=1015.968,-1.901,-118.956,-24.169,21.528,-42.882
C09979=1015.968,-1.489,-118.991,-24.170,21.527,-42.877
C09980=1015.967,-1.078,-119.025,-24.171,21.527,-42.872
C09981=1015.967,-0.671,-119.060,-24.171,21.526,-42.867
C09982=1015.966,-0.265,-119.094,-24.172,21.525,-42.862
C09983=1015.966,0.139,-119.128,-24.173,21.525,-42.857
C09984=1015.965,0.540,-119.163,-24.173,21.525,-42.851
C09985=1015.964,0.940,-119.197,-24.174,21.525,-42.846
C09986=1015.964,1.339,-119.230,-24.175,21.523,-42.841
C09987=1015.963,1.738,-119.264,-24.175,21.524,-42.836
C09988=1015.963,2.122,-119.296,-24.176,21.523,-42.833
C09989=1015.962,2.476,-119.326,-24.177,21.522,-42.827
C09990=1015.961,2.798,-119.353,-24.177,21.522,-42.823
C09991=1015.960,3.112,-119.380,-24.178,21.521,-42.817
C09992=1015.960,3.440,-119.408,-24.179,21.521,-42.812
C09993=1015.959,3.799,-119.438,-24.179,21.521,-42.809
C09994=1015.959,4.188,-119.471,-24.180,21.520,-42.805
C09995=1015.958,4.584,-119.505,-24.180,21.519,-42.799
C09996=1015.957,4.979,-119.539,-24.181,21.520,-42.794
//INST
///DATE 2021/06/17 16:00
///ATTR SC,RW,RJ
////FRAME ROBOT
///GROUP1 RB1
NOP
MOVL C00000 V=800.0 PL=0
MOVL C00001 V=800.0 PL=0
MOVL C00002 V=800.0 PL=0
MOVL C00003 V=800.0 PL=0
MOVL C00004 V=800.0 PL=0
MOVL C00005 V=800.0 PL=0
MOVL C00006 V=800.0 PL=0
MOVL C00007 V=800.0 PL=0
MOVL C00008 V=800.0 PL=0
MOVL C00009 V=800.0 PL=0
MOVL C00010 V=800.0 PL=0
MOVL C00011 V=800.0 PL=0
MOVL C00012 V=800.0 PL=0
MOVL C00013 V=800.0 PL=0
MOVL C00014 V=800.0 PL=0
MOVL C00015 V=800.0 PL=0
MOVL C00016 V=800.0 PL=0
MOVL C00017 V=800.0 PL=0
MOVL C00018 V=800.0 PL=0
MOVL C00019 V=800.0 PL=0
MOVL C00020 V=800.0 PL=0
MOVL C00021 V=800.0 PL=0
MOVL C00022 V=800.0 PL=0
MOVL C00023 V=800.0 PL=0
MOVL C00024 V=800.0 PL=0
MOVL C00025 V=800.0 PL=0
MOVL C00026 V=800.0 PL=0
MOVL C00027 V=800.0 PL=0
MOVL C00028 V=800.0 PL=0
MOVL C00029 V=800.0 PL=0
MOVL C00030 V=800.0 PL=0
MOVL C00031 V=800.0 PL=0
MOVL C00032 V=800.0 PL=0
MOVL C00033 V=800.0 PL=0
MOVL C00034 V=800.0 PL=0
MOVL C00035 V=800.0 PL=0
MOVL C00036 V=800.0 PL=0
MOVL C00037 V=800.0 PL=0
MOVL C00038 V=800.0 PL=0
MOVL C00039 V=800.0 PL=0
MOVL C00040 V=800.0 PL=0
MOVL C00041 V=800.0 PL=0
MOVL C00042 V=800.0 PL=0
MOVL C00043 V=800.0 PL=0
MOVL C00044 V=800.0 PL=0
MOVL C00045 V=800.0 PL=0
MOVL C00046 V=800.0 PL=0
MOVL C00047 V=800.0 PL=0
MOVL C00048 V=800.0 PL=0
MOVL C00049 V=800.0 PL=0
MOVL C00050 V=800.0 PL=0
MOVL C00051 V=800.0 PL=0
MOVL C00052 V=800.0 PL=0
MOVL C00053 V=800.0 PL=0
MOVL C00054 V=800.0 PL=0
MOVL C00055 V=800.0 PL=0
MOVL C00056 V=800.0 PL=0
MOVL C00057 V=800.0 PL=0
MOVL C00058 V=800.0 PL=0
MOVL C00059 V=800.0 PL=0
MOVL C00060 V=800.0 PL=0
MOVL C00061 V=800.0 PL=0
MOVL C00062 V=800.0 PL=0
MOVL C00063 V=800.0 PL=0
MOVL C00064 V=800.0 PL=0
MOVL C00065 V=800.0 PL=0
MOVL C00066 V=800.0 PL=0
MOVL C00067 V=800.0 PL=0
MOVL C00068 V=800.0 PL=0
MOVL C00069 V=800.0 PL=0
MOVL C00070 V=800.0 PL=0
MOVL C00071 V=800.0 PL=0
MOVL C00072 V=800.0 PL=0
MOVL C00073 V=800.0 PL=0
MOVL C00074 V=800.0 PL=0
MOVL C00075 V=800.0 PL=0
MOVL C00076 V=800.0 PL=0
MOVL C00077 V=800.0 PL=0
MOVL C00078 V=800.0 PL=0
MOVL C00079 V=800.0 PL=0
MOVL C00080 V=800.0 PL=0
MOVL C00081 V=800.0 PL=0
MOVL C00082 V=800.0 PL=0
MOVL C00083 V=800.0 PL=0
MOVL C00084 V=800.0 PL=0
MOVL C00085 V=800.0 PL=0
MOVL C00086 V=800.0 PL=0
MOVL C00087 V=800.0 PL=0
MOVL C00088 V=800.0 PL=0
MOVL C00089 V=800.0 PL=0
MOVL C00090 V=800.0 PL=0
MOVL C00091 V=800.0 PL=0
MOVL C00092 V=800.0 PL=0
MOVL C00093 V=800.0 PL=0
MOVL C00094 V=800.0 PL=0
MOVL C00095 V=800.0 PL=0
MOVL C00096 V=800.0 PL=0
MOVL C00097 V=800.0 PL=0
MOVL C00098 V=800.0 PL=0
MOVL C00099 V=800.0 PL=0
MOVL C00100 V=800.0 PL=0
MOVL C00101 V=800.0 PL=0
MOVL C00102 V=800.0 PL=0
MOVL C00103 V=800.0 PL=0
MOVL C00104 V=800.0 PL=0
MOVL C00105 V=800.0 PL=0
MOVL C00106 V=800.0 PL=0
MOVL C00107 V=800.0 PL=0
MOVL C00108 V=800.0 PL=0
MOVL C00109 V=800.0 PL=0
MOVL C00110 V=800.0 PL=0
MOVL C00111 V=800.0 PL=0
MOVL C00112 V=800.0 PL=0
MOVL C00113 V=800.0 PL=0
MOVL C00114 V=800.0 PL=0
MOVL C00115 V=800.0 PL=0
MOVL C00116 V=800.0 PL=0
MOVL C00117 V=800.0 PL=0
MOVL C00118 V=800.0 PL=0
MOVL C00119 V=800.0 PL=0
MOVL C00120 V=800.0 PL=0
MOVL C00121 V=800.0 PL=0
MOVL C00122 V=800.0 PL=0
MOVL C00123 V=800.0 PL=0
MOVL C00124 V=800.0 PL=0
MOVL C00125 V=800.0 PL=0
MOVL C00126 V=800.0 PL=0
MOVL C00127 V=800.0 PL=0
MOVL C00128 V=800.0 PL=0
MOVL C00129 V=800.0 PL=0
MOVL C00130 V=800.0 PL=0
MOVL C00131 V=800.0 PL=0
MOVL C00132 V=800.0 PL=0
MOVL C00133 V=800.0 PL=0
MOVL C00134 V=800.0 PL=0
MOVL C00135 V=800.0 PL=0
MOVL C00136 V=800.0 PL=0
MOVL C00137 V=800.0 PL=0
MOVL C00138 V=800.0 PL=0
MOVL C00139 V=800.0 PL=0
MOVL C00140 V=800.0 PL=0
MOVL C00141 V=800.0 PL=0
MOVL C00142 V=800.0 PL=0
MOVL C00143 V=800.0 PL=0
MOVL C00144 V=800.0 PL=0
MOVL C00145 V=800.0 PL=0
MOVL C00146 V=800.0 PL=0
MOVL C00147 V=800.0 PL=0
MOVL C00148 V=800.0 PL=0
MOVL C00149 V=800.0 PL=0
MOVL C00150 V=800.0 PL=0
MOVL C00151 V=800.0 PL=0
MOVL C00152 V=800.0 PL=0
MOVL C00153 V=800.0 PL=0
MOVL C00154 V=800.0 PL=0
MOVL C00155 V=800.0 PL=0
MOVL C00156 V=800.0 PL=0
MOVL C00157 V=800.0 PL=0
MOVL C00158 V=800.0 PL=0
MOVL C00159 V=800.0 PL=0
MOVL C00160 V=800.0 PL=0
MOVL C00161 V=800.0 PL=0
MOVL C00162 V=800.0 PL=0
MOVL C00163 V=800.0 PL=0
MOVL C00164 V=800.0 PL=0
MOVL C00165 V=800.0 PL=0
MOVL C00166 V=800.0 PL=0
MOVL C00167 V=800.0 PL=0
MOVL C00168 V=800.0 PL=0
MOVL C00169 V=800.0 PL=0
MOVL C00170 V=800.0 PL=0
MOVL C00171 V=800.0 PL=0
MOVL C00172 V=800.0 PL=0
MOVL C00173 V=800.0 PL=0
MOVL C00174 V=800.0 PL=0
MOVL C00175 V=800.0 PL=0
MOVL C00176 V=800.0 PL=0
MOVL C00177 V=800.0 PL=0
MOVL C00178 V=800.0 PL=0
MOVL C00179 V=800.0 PL=0
MOVL C00180 V=800.0 PL=0
MOVL C00181 V=800.0 PL=0
MOVL C00182 V=800.0 PL=0
MOVL C00183 V=800.0 PL=0
MOVL C00184 V=800.0 PL=0
MOVL C00185 V=800.0 PL=0
MOVL C00186 V=800.0 PL=0
MOVL C00187 V=800.0 PL=0
MOVL C00188 V=800.0 PL=0
MOVL C00189 V=800.0 PL=0
MOVL C00190 V=800.0 PL=0
MOVL C00191 V=800.0 PL=0
MOVL C00192 V=800.0 PL=0
MOVL C00193 V=800.0 PL=0
MOVL C00194 V=800.0 PL=0
MOVL C00195 V=800.0 PL=0
MOVL C00196 V=800.0 PL=0
MOVL C00197 V=800.0 PL=0
MOVL C00198 V=800.0 PL=0
MOVL C00199 V=800.0 PL=0
MOVL C00200 V=800.0 PL=0
MOVL C00201 V=800.0 PL=0
MOVL C00202 V=800.0 PL=0
MOVL C00203 V=800.0 PL=0
MOVL C00204 V=800.0 PL=0
MOVL C00205 V=800.0 PL=0
MOVL C00206 V=800.0 PL=0
MOVL C00207 V=800.0 PL=0
MOVL C00208 V=800.0 PL=0
MOVL C00209 V=800.0 PL=0
MOVL C00210 V=800.0 PL=0
MOVL C00211 V=800.0 PL=0
MOVL C00212 V=800.0 PL=0
MOVL C00213 V=800.0 PL=0
MOVL C00214 V=800.0 PL=0
MOVL C00215 V=800.0 PL=0
MOVL C00216 V=800.0 PL=0
MOVL C00217 V=800.0 PL=0
MOVL C00218 V=800.0 PL=0
MOVL C00219 V=800.0 PL=0
MOVL C00220 V=800.0 PL=0
MOVL C00221 V=800.0 PL=0
MOVL C00222 V=800.0 PL=0
MOVL C00223 V=800.0 PL=0
MOVL C00224 V=800.0 PL=0
MOVL C00225 V=800.0 PL=0
MOVL C00226 V=800.0 PL=0
MOVL C00227 V=800.0 PL=0
MOVL C00228 V=800.0 PL=0
MOVL C00229 V=800.0 PL=0
MOVL C00230 V=800.0 PL=0
MOVL C00231 V=800.0 PL=0
MOVL C00232 V=800.0 PL=0
MOVL C00233 V=800.0 PL=0
MOVL C00234 V=800.0 PL=0
MOVL C00235 V=800.0 PL=0
MOVL C00236 V=800.0 PL=0
MOVL C00237 V=800.0 PL=0
MOVL C00238 V=800.0 PL=0
MOVL C00239 V=800.0 PL=0
MOVL C00240 V=800.0 PL=0
MOVL C00241 V=800.0 PL=0
MOVL C00242 V=800.0 PL=0
MOVL C00243 V=800.0 PL=0
MOVL C00244 V=800.0 PL=0
MOVL C00245 V=800.0 PL=0
MOVL C00246 V=800.0 PL=0
MOVL C00247 V=800.0 PL=0
MOVL C00248 V=800.0 PL=0
MOVL C00249 V=800.0 PL=0
MOVL C00250 V=800.0 PL=0
MOVL C00251 V=800.0 PL=0
MOVL C00252 V=800.0 PL=0
MOVL C00253 V=800.0 PL=0
MOVL C00254 V=800.0 PL=0
MOVL C00255 V=800.0 PL=0
MOVL C00256 V=800.0 PL=0
MOVL C00257 V=800.0 PL=0
MOVL C00258 V=800.0 PL=0
MOVL C00259 V=800.0 PL=0
MOVL C00260 V=800.0 PL=0
MOVL C00261 V=800.0 PL=0
MOVL C00262 V=800.0 PL=0
MOVL C00263 V=800.0 PL=0
MOVL C00264 V=800.0 PL=0
MOVL C00265 V=800.0 PL=0
MOVL C00266 V=800.0 PL=0
MOVL C00267 V=800.0 PL=0
MOVL C00268 V=800.0 PL=0
MOVL C00269 V=800.0 PL=0
MOVL C00270 V=800.0 PL=0
MOVL C00271 V=800.0 PL=0
MOVL C00272 V=800.0 PL=0
MOVL C00273 V=800.0 PL=0
MOVL C00274 V=800.0 PL=0
MOVL C00275 V=800.0 PL=0
MOVL C00276 V=800.0 PL=0
MOVL C00277 V=800.0 PL=0
MOVL C00278 V=800.0 PL=0
MOVL C00279 V=800.0 PL=0
MOVL C00280 V=800.0 PL=0
MOVL C00281 V=800.0 PL=0
MOVL C00282 V=800.0 PL=0
MOVL C00283 V=800.0 PL=0
MOVL C00284 V=800.0 PL=0
MOVL C00285 V=800.0 PL=0
MOVL C00286 V=800.0 PL=0
MOVL C00287 V=800.0 PL=0
MOVL C00288 V=800.0 PL=0
MOVL C00289 V=800.0 PL=0
MOVL C00290 V=800.0 PL=0
MOVL C00291 V=800.0 PL=0
MOVL C00292 V=800.0 PL=0
MOVL C00293 V=800.0 PL=0
MOVL C00294 V=800.0 PL=0
MOVL C00295 V=800.0 PL=0
MOVL C00296 V=800.0 PL=0
MOVL C00297 V=800.0 PL=0
MOVL C00298 V=800.0 PL=0
MOVL C00299 V=800.0 PL=0
MOVL C00300 V=800.0 PL=0
MOVL C00301 V=800.0 PL=0
MOVL C00302 V=800.0 PL=0
MOVL C00303 V=800.0 PL=0
MOVL C00304 V=800.0 PL=0
MOVL C00305 V=800.0 PL=0
MOVL C00306 V=800.0 PL=0
MOVL C00307 V=800.0 PL=0
MOVL C00308 V=800.0 PL=0
MOVL C00309 V=800.0 PL=0
MOVL C00310 V=800.0 PL=0
MOVL C00311 V=800.0 PL=0
MOVL C00312 V=800.0 PL=0
MOVL C00313 V=800.0 PL=0
MOVL C00314 V=800.0 PL=0
MOVL C00315 V=800.0 PL=0
MOVL C00316 V=800.0 PL=0
MOVL C00317 V=800.0 PL=0
MOVL C00318 V=800.0 PL=0
MOVL C00319 V=800.0 PL=0
MOVL C00320 V=800.0 PL=0
MOVL C00321 V=800.0 PL=0
MOVL C00322 V=800.0 PL=0
MOVL C00323 V=800.0 PL=0
MOVL C00324 V=800.0 PL=0
MOVL C00325 V=800.0 PL=0
MOVL C00326 V=800.0 PL=0
MOVL C00327 V=800.0 PL=0
MOVL C00328 V=800.0 PL=0
MOVL C00329 V=800.0 PL=0
MOVL C00330 V=800.0 PL=0
MOVL C00331 V=800.0 PL=0
MOVL C00332 V=800.0 PL=0
MOVL C00333 V=800.0 PL=0
MOVL C00334 V=800.0 PL=0
MOVL C00335 V=800.0 PL=0
MOVL C00336 V=800.0 PL=0
MOVL C00337 V=800.0 PL=0
MOVL C00338 V=800.0 PL=0
MOVL C00339 V=800.0 PL=0
MOVL C00340 V=800.0 PL=0
MOVL C00341 V=800.0 PL=0
MOVL C00342 V=800.0 PL=0
MOVL C00343 V=800.0 PL=0
MOVL C00344 V=800.0 PL=0
MOVL C00345 V=800.0 PL=0
MOVL C00346 V=800.0 PL=0
MOVL C00347 V=800.0 PL=0
MOVL C00348 V=800.0 PL=0
MOVL C00349 V=800.0 PL=0
MOVL C00350 V=800.0 PL=0
MOVL C00351 V=800.0 PL=0
MOVL C00352 V=800.0 PL=0
MOVL C00353 V=800.0 PL=0
MOVL C00354 V=800.0 PL=0
MOVL C00355 V=800.0 PL=0
MOVL C00356 V=800.0 PL=0
MOVL C00357 V=800.0 PL=0
MOVL C00358 V=800.0 PL=0
MOVL C00359 V=800.0 PL=0
MOVL C00360 V=800.0 PL=0
MOVL C00361 V=800.0 PL=0
MOVL C00362 V=800.0 PL=0
MOVL C00363 V=800.0 PL=0
MOVL C00364 V=800.0 PL=0
MOVL C00365 V=800.0 PL=0
MOVL C00366 V=800.0 PL=0
MOVL C00367 V=800.0 PL=0
MOVL C00368 V=800.0 PL=0
MOVL C00369 V=800.0 PL=0
MOVL C00370 V=800.0 PL=0
MOVL C00371 V=800.0 PL=0
MOVL C00372 V=800.0 PL=0
MOVL C00373 V=800.0 PL=0
MOVL C00374 V=800.0 PL=0
MOVL C00375 V=800.0 PL=0
MOVL C00376 V=800.0 PL=0
MOVL C00377 V=800.0 PL=0
MOVL C00378 V=800.0 PL=0
MOVL C00379 V=800.0 PL=0
MOVL C00380 V=800.0 PL=0
MOVL C00381 V=800.0 PL=0
MOVL C00382 V=800.0 PL=0
MOVL C00383 V=800.0 PL=0
MOVL C00384 V=800.0 PL=0
MOVL C00385 V=800.0 PL=0
MOVL C00386 V=800.0 PL=0
MOVL C00387 V=800.0 PL=0
MOVL C00388 V=800.0 PL=0
MOVL C00389 V=800.0 PL=0
MOVL C00390 V=800.0 PL=0
MOVL C00391 V=800.0 PL=0
MOVL C00392 V=800.0 PL=0
MOVL C00393 V=800.0 PL=0
MOVL C00394 V=800.0 PL=0
MOVL C00395 V=800.0 PL=0
MOVL C00396 V=800.0 PL=0
MOVL C00397 V=800.0 PL=0
MOVL C00398 V=800.0 PL=0
MOVL C00399 V=800.0 PL=0
MOVL C00400 V=800.0 PL=0
MOVL C00401 V=800.0 PL=0
MOVL C00402 V=800.0 PL=0
MOVL C00403 V=800.0 PL=0
MOVL C00404 V=800.0 PL=0
MOVL C00405 V=800.0 PL=0
MOVL C00406 V=800.0 PL=0
MOVL C00407 V=800.0 PL=0
MOVL C00408 V=800.0 PL=0
MOVL C00409 V=800.0 PL=0
MOVL C00410 V=800.0 PL=0
MOVL C00411 V=800.0 PL=0
MOVL C00412 V=800.0 PL=0
MOVL C00413 V=800.0 PL=0
MOVL C00414 V=800.0 PL=0
MOVL C00415 V=800.0 PL=0
MOVL C00416 V=800.0 PL=0
MOVL C00417 V=800.0 PL=0
MOVL C00418 V=800.0 PL=0
MOVL C00419 V=800.0 PL=0
MOVL C00420 V=800.0 PL=0
MOVL C00421 V=800.0 PL=0
MOVL C00422 V=800.0 PL=0
MOVL C00423 V=800.0 PL=0
MOVL C00424 V=800.0 PL=0
MOVL C00425 V=800.0 PL=0
MOVL C00426 V=800.0 PL=0
MOVL C00427 V=800.0 PL=0
MOVL C00428 V=800.0 PL=0
MOVL C00429 V=800.0 PL=0
MOVL C00430 V=800.0 PL=0
MOVL C00431 V=800.0 PL=0
MOVL C00432 V=800.0 PL=0
MOVL C00433 V=800.0 PL=0
MOVL C00434 V=800.0 PL=0
MOVL C00435 V=800.0 PL=0
MOVL C00436 V=800.0 PL=0
MOVL C00437 V=800.0 PL=0
MOVL C00438 V=800.0 PL=0
MOVL C00439 V=800.0 PL=0
MOVL C00440 V=800.0 PL=0
MOVL C00441 V=800.0 PL=0
MOVL C00442 V=800.0 PL=0
MOVL C00443 V=800.0 PL=0
MOVL C00444 V=800.0 PL=0
MOVL C00445 V=800.0 PL=0
MOVL C00446 V=800.0 PL=0
MOVL C00447 V=800.0 PL=0
MOVL C00448 V=800.0 PL=0
MOVL C00449 V=800.0 PL=0
MOVL C00450 V=800.0 PL=0
MOVL C00451 V=800.0 PL=0
MOVL C00452 V=800.0 PL=0
MOVL C00453 V=800.0 PL=0
MOVL C00454 V=800.0 PL=0
MOVL C00455 V=800.0 PL=0
MOVL C00456 V=800.0 PL=0
MOVL C00457 V=800.0 PL=0
MOVL C00458 V=800.0 PL=0
MOVL C00459 V=800.0 PL=0
MOVL C00460 V=800.0 PL=0
MOVL C00461 V=800.0 PL=0
MOVL C00462 V=800.0 PL=0
MOVL C00463 V=800.0 PL=0
MOVL C00464 V=800.0 PL=0
MOVL C00465 V=800.0 PL=0
MOVL C00466 V=800.0 PL=0
MOVL C00467 V=800.0 PL=0
MOVL C00468 V=800.0 PL=0
MOVL C00469 V=800.0 PL=0
MOVL C00470 V=800.0 PL=0
MOVL C00471 V=800.0 PL=0
MOVL C00472 V=800.0 PL=0
MOVL C00473 V=800.0 PL=0
MOVL C00474 V=800.0 PL=0
MOVL C00475 V=800.0 PL=0
MOVL C00476 V=800.0 PL=0
MOVL C00477 V=800.0 PL=0
MOVL C00478 V=800.0 PL=0
MOVL C00479 V=800.0 PL=0
MOVL C00480 V=800.0 PL=0
MOVL C00481 V=800.0 PL=0
MOVL C00482 V=800.0 PL=0
MOVL C00483 V=800.0 PL=0
MOVL C00484 V=800.0 PL=0
MOVL C00485 V=800.0 PL=0
MOVL C00486 V=800.0 PL=0
MOVL C00487 V=800.0 PL=0
MOVL C00488 V=800.0 PL=0
MOVL C00489 V=800.0 PL=0
MOVL C00490 V=800.0 PL=0
MOVL C00491 V=800.0 PL=0
MOVL C00492 V=800.0 PL=0
MOVL C00493 V=800.0 PL=0
MOVL C00494 V=800.0 PL=0
MOVL C00495 V=800.0 PL=0
MOVL C00496 V=800.0 PL=0
MOVL C00497 V=800.0 PL=0
MOVL C00498 V=800.0 PL=0
MOVL C00499 V=800.0 PL=0
MOVL C00500 V=800.0 PL=0
MOVL C00501 V=800.0 PL=0
MOVL C00502 V=800.0 PL=0
MOVL C00503 V=800.0 PL=0
MOVL C00504 V=800.0 PL=0
MOVL C00505 V=800.0 PL=0
MOVL C00506 V=800.0 PL=0
MOVL C00507 V=800.0 PL=0
MOVL C00508 V=800.0 PL=0
MOVL C00509 V=800.0 PL=0
MOVL C00510 V=800.0 PL=0
MOVL C00511 V=800.0 PL=0
MOVL C00512 V=800.0 PL=0
MOVL C00513 V=800.0 PL=0
MOVL C00514 V=800.0 PL=0
MOVL C00515 V=800.0 PL=0
MOVL C00516 V=800.0 PL=0
MOVL C00517 V=800.0 PL=0
MOVL C00518 V=800.0 PL=0
MOVL C00519 V=800.0 PL=0
MOVL C00520 V=800.0 PL=0
MOVL C00521 V=800.0 PL=0
MOVL C00522 V=800.0 PL=0
MOVL C00523 V=800.0 PL=0
MOVL C00524 V=800.0 PL=0
MOVL C00525 V=800.0 PL=0
MOVL C00526 V=800.0 PL=0
MOVL C00527 V=800.0 PL=0
MOVL C00528 V=800.0 PL=0
MOVL C00529 V=800.0 PL=0
MOVL C00530 V=800.0 PL=0
MOVL C00531 V=800.0 PL=0
MOVL C00532 V=800.0 PL=0
MOVL C00533 V=800.0 PL=0
MOVL C00534 V=800.0 PL=0
MOVL C00535 V=800.0 PL=0
MOVL C00536 V=800.0 PL=0
MOVL C00537 V=800.0 PL=0
MOVL C00538 V=800.0 PL=0
MOVL C00539 V=800.0 PL=0
MOVL C00540 V=800.0 PL=0
MOVL C00541 V=800.0 PL=0
MOVL C00542 V=800.0 PL=0
MOVL C00543 V=800.0 PL=0
MOVL C00544 V=800.0 PL=0
MOVL C00545 V=800.0 PL=0
MOVL C00546 V=800.0 PL=0
MOVL C00547 V=800.0 PL=0
MOVL C00548 V=800.0 PL=0
MOVL C00549 V=800.0 PL=0
MOVL C00550 V=800.0 PL=0
MOVL C00551 V=800.0 PL=0
MOVL C00552 V=800.0 PL=0
MOVL C00553 V=800.0 PL=0
MOVL C00554 V=800.0 PL=0
MOVL C00555 V=800.0 PL=0
MOVL C00556 V=800.0 PL=0
MOVL C00557 V=800.0 PL=0
MOVL C00558 V=800.0 PL=0
MOVL C00559 V=800.0 PL=0
MOVL C00560 V=800.0 PL=0
MOVL C00561 V=800.0 PL=0
MOVL C00562 V=800.0 PL=0
MOVL C00563 V=800.0 PL=0
MOVL C00564 V=800.0 PL=0
MOVL C00565 V=800.0 PL=0
MOVL C00566 V=800.0 PL=0
MOVL C00567 V=800.0 PL=0
MOVL C00568 V=800.0 PL=0
MOVL C00569 V=800.0 PL=0
MOVL C00570 V=800.0 PL=0
MOVL C00571 V=800.0 PL=0
MOVL C00572 V=800.0 PL=0
MOVL C00573 V=800.0 PL=0
MOVL C00574 V=800.0 PL=0
MOVL C00575 V=800.0 PL=0
MOVL C00576 V=800.0 PL=0
MOVL C00577 V=800.0 PL=0
MOVL C00578 V=800.0 PL=0
MOVL C00579 V=800.0 PL=0
MOVL C00580 V=800.0 PL=0
MOVL C00581 V=800.0 PL=0
MOVL C00582 V=800.0 PL=0
MOVL C00583 V=800.0 PL=0
MOVL C00584 V=800.0 PL=0
MOVL C00585 V=800.0 PL=0
MOVL C00586 V=800.0 PL=0
MOVL C00587 V=800.0 PL=0
MOVL C00588 V=800.0 PL=0
MOVL C00589 V=800.0 PL=0
MOVL C00590 V=800.0 PL=0
MOVL C00591 V=800.0 PL=0
MOVL C00592 V=800.0 PL=0
MOVL C00593 V=800.0 PL=0
MOVL C00594 V=800.0 PL=0
MOVL C00595 V=800.0 PL=0
MOVL C00596 V=800.0 PL=0
MOVL C00597 V=800.0 PL=0
MOVL C00598 V=800.0 PL=0
MOVL C00599 V=800.0 PL=0
MOVL C00600 V=800.0 PL=0
MOVL C00601 V=800.0 PL=0
MOVL C00602 V=800.0 PL=0
MOVL C00603 V=800.0 PL=0
MOVL C00604 V=800.0 PL=0
MOVL C00605 V=800.0 PL=0
MOVL C00606 V=800.0 PL=0
MOVL C00607 V=800.0 PL=0
MOVL C00608 V=800.0 PL=0
MOVL C00609 V=800.0 PL=0
MOVL C00610 V=800.0 PL=0
MOVL C00611 V=800.0 PL=0
MOVL C00612 V=800.0 PL=0
MOVL C00613 V=800.0 PL=0
MOVL C00614 V=800.0 PL=0
MOVL C00615 V=800.0 PL=0
MOVL C00616 V=800.0 PL=0
MOVL C00617 V=800.0 PL=0
MOVL C00618 V=800.0 PL=0
MOVL C00619 V=800.0 PL=0
MOVL C00620 V=800.0 PL=0
MOVL C00621 V=800.0 PL=0
MOVL C00622 V=800.0 PL=0
MOVL C00623 V=800.0 PL=0
MOVL C00624 V=800.0 PL=0
MOVL C00625 V=800.0 PL=0
MOVL C00626 V=800.0 PL=0
MOVL C00627 V=800.0 PL=0
MOVL C00628 V=800.0 PL=0
MOVL C00629 V=800.0 PL=0
MOVL C00630 V=800.0 PL=0
MOVL C00631 V=800.0 PL=0
MOVL C00632 V=800.0 PL=0
MOVL C00633 V=800.0 PL=0
MOVL C00634 V=800.0 PL=0
MOVL C00635 V=800.0 PL=0
MOVL C00636 V=800.0 PL=0
MOVL C00637 V=800.0 PL=0
MOVL C00638 V=800.0 PL=0
MOVL C00639 V=800.0 PL=0
MOVL C00640 V=800.0 PL=0
MOVL C00641 V=800.0 PL=0
MOVL C00642 V=800.0 PL=0
MOVL C00643 V=800.0 PL=0
MOVL C00644 V=800.0 PL=0
MOVL C00645 V=800.0 PL=0
MOVL C00646 V=800.0 PL=0
MOVL C00647 V=800.0 PL=0
MOVL C00648 V=800.0 PL=0
MOVL C00649 V=800.0 PL=0
MOVL C00650 V=800.0 PL=0
MOVL C00651 V=800.0 PL=0
MOVL C00652 V=800.0 PL=0
MOVL C00653 V=800.0 PL=0
MOVL C00654 V=800.0 PL=0
MOVL C00655 V=800.0 PL=0
MOVL C00656 V=800.0 PL=0
MOVL C00657 V=800.0 PL=0
MOVL C00658 V=800.0 PL=0
MOVL C00659 V=800.0 PL=0
MOVL C00660 V=800.0 PL=0
MOVL C00661 V=800.0 PL=0
MOVL C00662 V=800.0 PL=0
MOVL C00663 V=800.0 PL=0
MOVL C00664 V=800.0 PL=0
MOVL C00665 V=800.0 PL=0
MOVL C00666 V=800.0 PL=0
MOVL C00667 V=800.0 PL=0
MOVL C00668 V=800.0 PL=0
MOVL C00669 V=800.0 PL=0
MOVL C00670 V=800.0 PL=0
MOVL C00671 V=800.0 PL=0
MOVL C00672 V=800.0 PL=0
MOVL C00673 V=800.0 PL=0
MOVL C00674 V=800.0 PL=0
MOVL C00675 V=800.0 PL=0
MOVL C00676 V=800.0 PL=0
MOVL C00677 V=800.0 PL=0
MOVL C00678 V=800.0 PL=0
MOVL C00679 V=800.0 PL=0
MOVL C00680 V=800.0 PL=0
MOVL C00681 V=800.0 PL=0
MOVL C00682 V=800.0 PL=0
MOVL C00683 V=800.0 PL=0
MOVL C00684 V=800.0 PL=0
MOVL C00685 V=800.0 PL=0
MOVL C00686 V=800.0 PL=0
MOVL C00687 V=800.0 PL=0
MOVL C00688 V=800.0 PL=0
MOVL C00689 V=800.0 PL=0
MOVL C00690 V=800.0 PL=0
MOVL C00691 V=800.0 PL=0
MOVL C00692 V=800.0 PL=0
MOVL C00693 V=800.0 PL=0
MOVL C00694 V=800.0 PL=0
MOVL C00695 V=800.0 PL=0
MOVL C00696 V=800.0 PL=0
MOVL C00697 V=800.0 PL=0
MOVL C00698 V=800.0 PL=0
MOVL C00699 V=800.0 PL=0
MOVL C00700 V=800.0 PL=0
MOVL C00701 V=800.0 PL=0
MOVL C00702 V=800.0 PL=0
MOVL C00703 V=800.0 PL=0
MOVL C00704 V=800.0 PL=0
MOVL C00705 V=800.0 PL=0
MOVL C00706 V=800.0 PL=0
MOVL C00707 V=800.0 PL=0
MOVL C00708 V=800.0 PL=0
MOVL C00709 V=800.0 PL=0
MOVL C00710 V=800.0 PL=0
MOVL C00711 V=800.0 PL=0
MOVL C00712 V=800.0 PL=0
MOVL C00713 V=800.0 PL=0
MOVL C00714 V=800.0 PL=0
MOVL C00715 V=800.0 PL=0
MOVL C00716 V=800.0 PL=0
MOVL C00717 V=800.0 PL=0
MOVL C00718 V=800.0 PL=0
MOVL C00719 V=800.0 PL=0
MOVL C00720 V=800.0 PL=0
MOVL C00721 V=800.0 PL=0
MOVL C00722 V=800.0 PL=0
MOVL C00723 V=800.0 PL=0
MOVL C00724 V=800.0 PL=0
MOVL C00725 V=800.0 PL=0
MOVL C00726 V=800.0 PL=0
MOVL C00727 V=800.0 PL=0
MOVL C00728 V=800.0 PL=0
MOVL C00729 V=800.0 PL=0
MOVL C00730 V=800.0 PL=0
MOVL C00731 V=800.0 PL=0
MOVL C00732 V=800.0 PL=0
MOVL C00733 V=800.0 PL=0
MOVL C00734 V=800.0 PL=0
MOVL C00735 V=800.0 PL=0
MOVL C00736 V=800.0 PL=0
MOVL C00737 V=800.0 PL=0
MOVL C00738 V=800.0 PL=0
MOVL C00739 V=800.0 PL=0
MOVL C00740 V=800.0 PL=0
MOVL C00741 V=800.0 PL=0
MOVL C00742 V=800.0 PL=0
MOVL C00743 V=800.0 PL=0
MOVL C00744 V=800.0 PL=0
MOVL C00745 V=800.0 PL=0
MOVL C00746 V=800.0 PL=0
MOVL C00747 V=800.0 PL=0
MOVL C00748 V=800.0 PL=0
MOVL C00749 V=800.0 PL=0
MOVL C00750 V=800.0 PL=0
MOVL C00751 V=800.0 PL=0
MOVL C00752 V=800.0 PL=0
MOVL C00753 V=800.0 PL=0
MOVL C00754 V=800.0 PL=0
MOVL C00755 V=800.0 PL=0
MOVL C00756 V=800.0 PL=0
MOVL C00757 V=800.0 PL=0
MOVL C00758 V=800.0 PL=0
MOVL C00759 V=800.0 PL=0
MOVL C00760 V=800.0 PL=0
MOVL C00761 V=800.0 PL=0
MOVL C00762 V=800.0 PL=0
MOVL C00763 V=800.0 PL=0
MOVL C00764 V=800.0 PL=0
MOVL C00765 V=800.0 PL=0
MOVL C00766 V=800.0 PL=0
MOVL C00767 V=800.0 PL=0
MOVL C00768 V=800.0 PL=0
MOVL C00769 V=800.0 PL=0
MOVL C00770 V=800.0 PL=0
MOVL C00771 V=800.0 PL=0
MOVL C00772 V=800.0 PL=0
MOVL C00773 V=800.0 PL=0
MOVL C00774 V=800.0 PL=0
MOVL C00775 V=800.0 PL=0
MOVL C00776 V=800.0 PL=0
MOVL C00777 V=800.0 PL=0
MOVL C00778 V=800.0 PL=0
MOVL C00779 V=800.0 PL=0
MOVL C00780 V=800.0 PL=0
MOVL C00781 V=800.0 PL=0
MOVL C00782 V=800.0 PL=0
MOVL C00783 V=800.0 PL=0
MOVL C00784 V=800.0 PL=0
MOVL C00785 V=800.0 PL=0
MOVL C00786 V=800.0 PL=0
MOVL C00787 V=800.0 PL=0
MOVL C00788 V=800.0 PL=0
MOVL C00789 V=800.0 PL=0
MOVL C00790 V=800.0 PL=0
MOVL C00791 V=800.0 PL=0
MOVL C00792 V=800.0 PL=0
MOVL C00793 V=800.0 PL=0
MOVL C00794 V=800.0 PL=0
MOVL C00795 V=800.0 PL=0
MOVL C00796 V=800.0 PL=0
MOVL C00797 V=800.0 PL=0
MOVL C00798 V=800.0 PL=0
MOVL C00799 V=800.0 PL=0
MOVL C00800 V=800.0 PL=0
MOVL C00801 V=800.0 PL=0
MOVL C00802 V=800.0 PL=0
MOVL C00803 V=800.0 PL=0
MOVL C00804 V=800.0 PL=0
MOVL C00805 V=800.0 PL=0
MOVL C00806 V=800.0 PL=0
MOVL C00807 V=800.0 PL=0
MOVL C00808 V=800.0 PL=0
MOVL C00809 V=800.0 PL=0
MOVL C00810 V=800.0 PL=0
MOVL C00811 V=800.0 PL=0
MOVL C00812 V=800.0 PL=0
MOVL C00813 V=800.0 PL=0
MOVL C00814 V=800.0 PL=0
MOVL C00815 V=800.0 PL=0
MOVL C00816 V=800.0 PL=0
MOVL C00817 V=800.0 PL=0
MOVL C00818 V=800.0 PL=0
MOVL C00819 V=800.0 PL=0
MOVL C00820 V=800.0 PL=0
MOVL C00821 V=800.0 PL=0
MOVL C00822 V=800.0 PL=0
MOVL C00823 V=800.0 PL=0
MOVL C00824 V=800.0 PL=0
MOVL C00825 V=800.0 PL=0
MOVL C00826 V=800.0 PL=0
MOVL C00827 V=800.0 PL=0
MOVL C00828 V=800.0 PL=0
MOVL C00829 V=800.0 PL=0
MOVL C00830 V=800.0 PL=0
MOVL C00831 V=800.0 PL=0
MOVL C00832 V=800.0 PL=0
MOVL C00833 V=800.0 PL=0
MOVL C00834 V=800.0 PL=0
MOVL C00835 V=800.0 PL=0
MOVL C00836 V=800.0 PL=0
MOVL C00837 V=800.0 PL=0
MOVL C00838 V=800.0 PL=0
MOVL C00839 V=800.0 PL=0
MOVL C00840 V=800.0 PL=0
MOVL C00841 V=800.0 PL=0
MOVL C00842 V=800.0 PL=0
MOVL C00843 V=800.0 PL=0
MOVL C00844 V=800.0 PL=0
MOVL C00845 V=800.0 PL=0
MOVL C00846 V=800.0 PL=0
MOVL C00847 V=800.0 PL=0
MOVL C00848 V=800.0 PL=0
MOVL C00849 V=800.0 PL=0
MOVL C00850 V=800.0 PL=0
MOVL C00851 V=800.0 PL=0
MOVL C00852 V=800.0 PL=0
MOVL C00853 V=800.0 PL=0
MOVL C00854 V=800.0 PL=0
MOVL C00855 V=800.0 PL=0
MOVL C00856 V=800.0 PL=0
MOVL C00857 V=800.0 PL=0
MOVL C00858 V=800.0 PL=0
MOVL C00859 V=800.0 PL=0
MOVL C00860 V=800.0 PL=0
MOVL C00861 V=800.0 PL=0
MOVL C00862 V=800.0 PL=0
MOVL C00863 V=800.0 PL=0
MOVL C00864 V=800.0 PL=0
MOVL C00865 V=800.0 PL=0
MOVL C00866 V=800.0 PL=0
MOVL C00867 V=800.0 PL=0
MOVL C00868 V=800.0 PL=0
MOVL C00869 V=800.0 PL=0
MOVL C00870 V=800.0 PL=0
MOVL C00871 V=800.0 PL=0
MOVL C00872 V=800.0 PL=0
MOVL C00873 V=800.0 PL=0
MOVL C00874 V=800.0 PL=0
MOVL C00875 V=800.0 PL=0
MOVL C00876 V=800.0 PL=0
MOVL C00877 V=800.0 PL=0
MOVL C00878 V=800.0 PL=0
MOVL C00879 V=800.0 PL=0
MOVL C00880 V=800.0 PL=0
MOVL C00881 V=800.0 PL=0
MOVL C00882 V=800.0 PL=0
MOVL C00883 V=800.0 PL=0
MOVL C00884 V=800.0 PL=0
MOVL C00885 V=800.0 PL=0
MOVL C00886 V=800.0 PL=0
MOVL C00887 V=800.0 PL=0
MOVL C00888 V=800.0 PL=0
MOVL C00889 V=800.0 PL=0
MOVL C00890 V=800.0 PL=0
MOVL C00891 V=800.0 PL=0
MOVL C00892 V=800.0 PL=0
MOVL C00893 V=800.0 PL=0
MOVL C00894 V=800.0 PL=0
MOVL C00895 V=800.0 PL=0
MOVL C00896 V=800.0 PL=0
MOVL C00897 V=800.0 PL=0
MOVL C00898 V=800.0 PL=0
MOVL C00899 V=800.0 PL=0
MOVL C00900 V=800.0 PL=0
MOVL C00901 V=800.0 PL=0
MOVL C00902 V=800.0 PL=0
MOVL C00903 V=800.0 PL=0
MOVL C00904 V=800.0 PL=0
MOVL C00905 V=800.0 PL=0
MOVL C00906 V=800.0 PL=0
MOVL C00907 V=800.0 PL=0
MOVL C00908 V=800.0 PL=0
MOVL C00909 V=800.0 PL=0
MOVL C00910 V=800.0 PL=0
MOVL C00911 V=800.0 PL=0
MOVL C00912 V=800.0 PL=0
MOVL C00913 V=800.0 PL=0
MOVL C00914 V=800.0 PL=0
MOVL C00915 V=800.0 PL=0
MOVL C00916 V=800.0 PL=0
MOVL C00917 V=800.0 PL=0
MOVL C00918 V=800.0 PL=0
MOVL C00919 V=800.0 PL=0
MOVL C00920 V=800.0 PL=0
MOVL C00921 V=800.0 PL=0
MOVL C00922 V=800.0 PL=0
MOVL C00923 V=800.0 PL=0
MOVL C00924 V=800.0 PL=0
MOVL C00925 V=800.0 PL=0
MOVL C00926 V=800.0 PL=0
MOVL C00927 V=800.0 PL=0
MOVL C00928 V=800.0 PL=0
MOVL C00929 V=800.0 PL=0
MOVL C00930 V=800.0 PL=0
MOVL C00931 V=800.0 PL=0
MOVL C00932 V=800.0 PL=0
MOVL C00933 V=800.0 PL=0
MOVL C00934 V=800.0 PL=0
MOVL C00935 V=800.0 PL=0
MOVL C00936 V=800.0 PL=0
MOVL C00937 V=800.0 PL=0
MOVL C00938 V=800.0 PL=0
MOVL C00939 V=800.0 PL=0
MOVL C00940 V=800.0 PL=0
MOVL C00941 V=800.0 PL=0
MOVL C00942 V=800.0 PL=0
MOVL C00943 V=800.0 PL=0
MOVL C00944 V=800.0 PL=0
MOVL C00945 V=800.0 PL=0
MOVL C00946 V=800.0 PL=0
MOVL C00947 V=800.0 PL=0
MOVL C00948 V=800.0 PL=0
MOVL C00949 V=800.0 PL=0
MOVL C00950 V=800.0 PL=0
MOVL C00951 V=800.0 PL=0
MOVL C00952 V=800.0 PL=0
MOVL C00953 V=800.0 PL=0
MOVL C00954 V=800.0 PL=0
MOVL C00955 V=800.0 PL=0
MOVL C00956 V=800.0 PL=0
MOVL C00957 V=800.0 PL=0
MOVL C00958 V=800.0 PL=0
MOVL C00959 V=800.0 PL=0
MOVL C00960 V=800.0 PL=0
MOVL C00961 V=800.0 PL=0
MOVL C00962 V=800.0 PL=0
MOVL C00963 V=800.0 PL=0
MOVL C00964 V=800.0 PL=0
MOVL C00965 V=800.0 PL=0
MOVL C00966 V=800.0 PL=0
MOVL C00967 V=800.0 PL=0
MOVL C00968 V=800.0 PL=0
MOVL C00969 V=800.0 PL=0
MOVL C00970 V=800.0 PL=0
MOVL C00971 V=800.0 PL=0
MOVL C00972 V=800.0 PL=0
MOVL C00973 V=800.0 PL=0
MOVL C00974 V=800.0 PL=0
MOVL C00975 V=800.0 PL=0
MOVL C00976 V=800.0 PL=0
MOVL C00977 V=800.0 PL=0
MOVL C00978 V=800.0 PL=0
MOVL C00979 V=800.0 PL=0
MOVL C00980 V=800.0 PL=0
MOVL C00981 V=800.0 PL=0
MOVL C00982 V=800.0 PL=0
MOVL C00983 V=800.0 PL=0
MOVL C00984 V=800.0 PL=0
MOVL C00985 V=800.0 PL=0
MOVL C00986 V=800.0 PL=0
MOVL C00987 V=800.0 PL=0
MOVL C00988 V=800.0 PL=0
MOVL C00989 V=800.0 PL=0
MOVL C00990 V=800.0 PL=0
MOVL C00991 V=800.0 PL=0
MOVL C00992 V=800.0 PL=0
MOVL C00993 V=800.0 PL=0
MOVL C00994 V=800.0 PL=0
MOVL C00995 V=800.0 PL=0
MOVL C00996 V=800.0 PL=0
MOVL C00997 V=800.0 PL=0
MOVL C00998 V=800.0 PL=0
MOVL C00999 V=800.0 PL=0
MOVL C01000 V=800.0 PL=0
MOVL C01001 V=800.0 PL=0
MOVL C01002 V=800.0 PL=0
MOVL C01003 V=800.0 PL=0
MOVL C01004 V=800.0 PL=0
MOVL C01005 V=800.0 PL=0
MOVL C01006 V=800.0 PL=0
MOVL C01007 V=800.0 PL=0
MOVL C01008 V=800.0 PL=0
MOVL C01009 V=800.0 PL=0
MOVL C01010 V=800.0 PL=0
MOVL C01011 V=800.0 PL=0
MOVL C01012 V=800.0 PL=0
MOVL C01013 V=800.0 PL=0
MOVL C01014 V=800.0 PL=0
MOVL C01015 V=800.0 PL=0
MOVL C01016 V=800.0 PL=0
MOVL C01017 V=800.0 PL=0
MOVL C01018 V=800.0 PL=0
MOVL C01019 V=800.0 PL=0
MOVL C01020 V=800.0 PL=0
MOVL C01021 V=800.0 PL=0
MOVL C01022 V=800.0 PL=0
MOVL C01023 V=800.0 PL=0
MOVL C01024 V=800.0 PL=0
MOVL C01025 V=800.0 PL=0
MOVL C01026 V=800.0 PL=0
MOVL C01027 V=800.0 PL=0
MOVL C01028 V=800.0 PL=0
MOVL C01029 V=800.0 PL=0
MOVL C01030 V=800.0 PL=0
MOVL C01031 V=800.0 PL=0
MOVL C01032 V=800.0 PL=0
MOVL C01033 V=800.0 PL=0
MOVL C01034 V=800.0 PL=0
MOVL C01035 V=800.0 PL=0
MOVL C01036 V=800.0 PL=0
MOVL C01037 V=800.0 PL=0
MOVL C01038 V=800.0 PL=0
MOVL C01039 V=800.0 PL=0
MOVL C01040 V=800.0 PL=0
MOVL C01041 V=800.0 PL=0
MOVL C01042 V=800.0 PL=0
MOVL C01043 V=800.0 PL=0
MOVL C01044 V=800.0 PL=0
MOVL C01045 V=800.0 PL=0
MOVL C01046 V=800.0 PL=0
MOVL C01047 V=800.0 PL=0
MOVL C01048 V=800.0 PL=0
MOVL C01049 V=800.0 PL=0
MOVL C01050 V=800.0 PL=0
MOVL C01051 V=800.0 PL=0
MOVL C01052 V=800.0 PL=0
MOVL C01053 V=800.0 PL=0
MOVL C01054 V=800.0 PL=0
MOVL C01055 V=800.0 PL=0
MOVL C01056 V=800.0 PL=0
MOVL C01057 V=800.0 PL=0
MOVL C01058 V=800.0 PL=0
MOVL C01059 V=800.0 PL=0
MOVL C01060 V=800.0 PL=0
MOVL C01061 V=800.0 PL=0
MOVL C01062 V=800.0 PL=0
MOVL C01063 V=800.0 PL=0
MOVL C01064 V=800.0 PL=0
MOVL C01065 V=800.0 PL=0
MOVL C01066 V=800.0 PL=0
MOVL C01067 V=800.0 PL=0
MOVL C01068 V=800.0 PL=0
MOVL C01069 V=800.0 PL=0
MOVL C01070 V=800.0 PL=0
MOVL C01071 V=800.0 PL=0
MOVL C01072 V=800.0 PL=0
MOVL C01073 V=800.0 PL=0
MOVL C01074 V=800.0 PL=0
MOVL C01075 V=800.0 PL=0
MOVL C01076 V=800.0 PL=0
MOVL C01077 V=800.0 PL=0
MOVL C01078 V=800.0 PL=0
MOVL C01079 V=800.0 PL=0
MOVL C01080 V=800.0 PL=0
MOVL C01081 V=800.0 PL=0
MOVL C01082 V=800.0 PL=0
MOVL C01083 V=800.0 PL=0
MOVL C01084 V=800.0 PL=0
MOVL C01085 V=800.0 PL=0
MOVL C01086 V=800.0 PL=0
MOVL C01087 V=800.0 PL=0
MOVL C01088 V=800.0 PL=0
MOVL C01089 V=800.0 PL=0
MOVL C01090 V=800.0 PL=0
MOVL C01091 V=800.0 PL=0
MOVL C01092 V=800.0 PL=0
MOVL C01093 V=800.0 PL=0
MOVL C01094 V=800.0 PL=0
MOVL C01095 V=800.0 PL=0
MOVL C01096 V=800.0 PL=0
MOVL C01097 V=800.0 PL=0
MOVL C01098 V=800.0 PL=0
MOVL C01099 V=800.0 PL=0
MOVL C01100 V=800.0 PL=0
MOVL C01101 V=800.0 PL=0
MOVL C01102 V=800.0 PL=0
MOVL C01103 V=800.0 PL=0
MOVL C01104 V=800.0 PL=0
MOVL C01105 V=800.0 PL=0
MOVL C01106 V=800.0 PL=0
MOVL C01107 V=800.0 PL=0
MOVL C01108 V=800.0 PL=0
MOVL C01109 V=800.0 PL=0
MOVL C01110 V=800.0 PL=0
MOVL C01111 V=800.0 PL=0
MOVL C01112 V=800.0 PL=0
MOVL C01113 V=800.0 PL=0
MOVL C01114 V=800.0 PL=0
MOVL C01115 V=800.0 PL=0
MOVL C01116 V=800.0 PL=0
MOVL C01117 V=800.0 PL=0
MOVL C01118 V=800.0 PL=0
MOVL C01119 V=800.0 PL=0
MOVL C01120 V=800.0 PL=0
MOVL C01121 V=800.0 PL=0
MOVL C01122 V=800.0 PL=0
MOVL C01123 V=800.0 PL=0
MOVL C01124 V=800.0 PL=0
MOVL C01125 V=800.0 PL=0
MOVL C01126 V=800.0 PL=0
MOVL C01127 V=800.0 PL=0
MOVL C01128 V=800.0 PL=0
MOVL C01129 V=800.0 PL=0
MOVL C01130 V=800.0 PL=0
MOVL C01131 V=800.0 PL=0
MOVL C01132 V=800.0 PL=0
MOVL C01133 V=800.0 PL=0
MOVL C01134 V=800.0 PL=0
MOVL C01135 V=800.0 PL=0
MOVL C01136 V=800.0 PL=0
MOVL C01137 V=800.0 PL=0
MOVL C01138 V=800.0 PL=0
MOVL C01139 V=800.0 PL=0
MOVL C01140 V=800.0 PL=0
MOVL C01141 V=800.0 PL=0
MOVL C01142 V=800.0 PL=0
MOVL C01143 V=800.0 PL=0
MOVL C01144 V=800.0 PL=0
MOVL C01145 V=800.0 PL=0
MOVL C01146 V=800.0 PL=0
MOVL C01147 V=800.0 PL=0
MOVL C01148 V=800.0 PL=0
MOVL C01149 V=800.0 PL=0
MOVL C01150 V=800.0 PL=0
MOVL C01151 V=800.0 PL=0
MOVL C01152 V=800.0 PL=0
MOVL C01153 V=800.0 PL=0
MOVL C01154 V=800.0 PL=0
MOVL C01155 V=800.0 PL=0
MOVL C01156 V=800.0 PL=0
MOVL C01157 V=800.0 PL=0
MOVL C01158 V=800.0 PL=0
MOVL C01159 V=800.0 PL=0
MOVL C01160 V=800.0 PL=0
MOVL C01161 V=800.0 PL=0
MOVL C01162 V=800.0 PL=0
MOVL C01163 V=800.0 PL=0
MOVL C01164 V=800.0 PL=0
MOVL C01165 V=800.0 PL=0
MOVL C01166 V=800.0 PL=0
MOVL C01167 V=800.0 PL=0
MOVL C01168 V=800.0 PL=0
MOVL C01169 V=800.0 PL=0
MOVL C01170 V=800.0 PL=0
MOVL C01171 V=800.0 PL=0
MOVL C01172 V=800.0 PL=0
MOVL C01173 V=800.0 PL=0
MOVL C01174 V=800.0 PL=0
MOVL C01175 V=800.0 PL=0
MOVL C01176 V=800.0 PL=0
MOVL C01177 V=800.0 PL=0
MOVL C01178 V=800.0 PL=0
MOVL C01179 V=800.0 PL=0
MOVL C01180 V=800.0 PL=0
MOVL C01181 V=800.0 PL=0
MOVL C01182 V=800.0 PL=0
MOVL C01183 V=800.0 PL=0
MOVL C01184 V=800.0 PL=0
MOVL C01185 V=800.0 PL=0
MOVL C01186 V=800.0 PL=0
MOVL C01187 V=800.0 PL=0
MOVL C01188 V=800.0 PL=0
MOVL C01189 V=800.0 PL=0
MOVL C01190 V=800.0 PL=0
MOVL C01191 V=800.0 PL=0
MOVL C01192 V=800.0 PL=0
MOVL C01193 V=800.0 PL=0
MOVL C01194 V=800.0 PL=0
MOVL C01195 V=800.0 PL=0
MOVL C01196 V=800.0 PL=0
MOVL C01197 V=800.0 PL=0
MOVL C01198 V=800.0 PL=0
MOVL C01199 V=800.0 PL=0
MOVL C01200 V=800.0 PL=0
MOVL C01201 V=800.0 PL=0
MOVL C01202 V=800.0 PL=0
MOVL C01203 V=800.0 PL=0
MOVL C01204 V=800.0 PL=0
MOVL C01205 V=800.0 PL=0
MOVL C01206 V=800.0 PL=0
MOVL C01207 V=800.0 PL=0
MOVL C01208 V=800.0 PL=0
MOVL C01209 V=800.0 PL=0
MOVL C01210 V=800.0 PL=0
MOVL C01211 V=800.0 PL=0
MOVL C01212 V=800.0 PL=0
MOVL C01213 V=800.0 PL=0
MOVL C01214 V=800.0 PL=0
MOVL C01215 V=800.0 PL=0
MOVL C01216 V=800.0 PL=0
MOVL C01217 V=800.0 PL=0
MOVL C01218 V=800.0 PL=0
MOVL C01219 V=800.0 PL=0
MOVL C01220 V=800.0 PL=0
MOVL C01221 V=800.0 PL=0
MOVL C01222 V=800.0 PL=0
MOVL C01223 V=800.0 PL=0
MOVL C01224 V=800.0 PL=0
MOVL C01225 V=800.0 PL=0
MOVL C01226 V=800.0 PL=0
MOVL C01227 V=800.0 PL=0
MOVL C01228 V=800.0 PL=0
MOVL C01229 V=800.0 PL=0
MOVL C01230 V=800.0 PL=0
MOVL C01231 V=800.0 PL=0
MOVL C01232 V=800.0 PL=0
MOVL C01233 V=800.0 PL=0
MOVL C01234 V=800.0 PL=0
MOVL C01235 V=800.0 PL=0
MOVL C01236 V=800.0 PL=0
MOVL C01237 V=800.0 PL=0
MOVL C01238 V=800.0 PL=0
MOVL C01239 V=800.0 PL=0
MOVL C01240 V=800.0 PL=0
MOVL C01241 V=800.0 PL=0
MOVL C01242 V=800.0 PL=0
MOVL C01243 V=800.0 PL=0
MOVL C01244 V=800.0 PL=0
MOVL C01245 V=800.0 PL=0
MOVL C01246 V=800.0 PL=0
MOVL C01247 V=800.0 PL=0
MOVL C01248 V=800.0 PL=0
MOVL C01249 V=800.0 PL=0
MOVL C01250 V=800.0 PL=0
MOVL C01251 V=800.0 PL=0
MOVL C01252 V=800.0 PL=0
MOVL C01253 V=800.0 PL=0
MOVL C01254 V=800.0 PL=0
MOVL C01255 V=800.0 PL=0
MOVL C01256 V=800.0 PL=0
MOVL C01257 V=800.0 PL=0
MOVL C01258 V=800.0 PL=0
MOVL C01259 V=800.0 PL=0
MOVL C01260 V=800.0 PL=0
MOVL C01261 V=800.0 PL=0
MOVL C01262 V=800.0 PL=0
MOVL C01263 V=800.0 PL=0
MOVL C01264 V=800.0 PL=0
MOVL C01265 V=800.0 PL=0
MOVL C01266 V=800.0 PL=0
MOVL C01267 V=800.0 PL=0
MOVL C01268 V=800.0 PL=0
MOVL C01269 V=800.0 PL=0
MOVL C01270 V=800.0 PL=0
MOVL C01271 V=800.0 PL=0
MOVL C01272 V=800.0 PL=0
MOVL C01273 V=800.0 PL=0
MOVL C01274 V=800.0 PL=0
MOVL C01275 V=800.0 PL=0
MOVL C01276 V=800.0 PL=0
MOVL C01277 V=800.0 PL=0
MOVL C01278 V=800.0 PL=0
MOVL C01279 V=800.0 PL=0
MOVL C01280 V=800.0 PL=0
MOVL C01281 V=800.0 PL=0
MOVL C01282 V=800.0 PL=0
MOVL C01283 V=800.0 PL=0
MOVL C01284 V=800.0 PL=0
MOVL C01285 V=800.0 PL=0
MOVL C01286 V=800.0 PL=0
MOVL C01287 V=800.0 PL=0
MOVL C01288 V=800.0 PL=0
MOVL C01289 V=800.0 PL=0
MOVL C01290 V=800.0 PL=0
MOVL C01291 V=800.0 PL=0
MOVL C01292 V=800.0 PL=0
MOVL C01293 V=800.0 PL=0
MOVL C01294 V=800.0 PL=0
MOVL C01295 V=800.0 PL=0
MOVL C01296 V=800.0 PL=0
MOVL C01297 V=800.0 PL=0
MOVL C01298 V=800.0 PL=0
MOVL C01299 V=800.0 PL=0
MOVL C01300 V=800.0 PL=0
MOVL C01301 V=800.0 PL=0
MOVL C01302 V=800.0 PL=0
MOVL C01303 V=800.0 PL=0
MOVL C01304 V=800.0 PL=0
MOVL C01305 V=800.0 PL=0
MOVL C01306 V=800.0 PL=0
MOVL C01307 V=800.0 PL=0
MOVL C01308 V=800.0 PL=0
MOVL C01309 V=800.0 PL=0
MOVL C01310 V=800.0 PL=0
MOVL C01311 V=800.0 PL=0
MOVL C01312 V=800.0 PL=0
MOVL C01313 V=800.0 PL=0
MOVL C01314 V=800.0 PL=0
MOVL C01315 V=800.0 PL=0
MOVL C01316 V=800.0 PL=0
MOVL C01317 V=800.0 PL=0
MOVL C01318 V=800.0 PL=0
MOVL C01319 V=800.0 PL=0
MOVL C01320 V=800.0 PL=0
MOVL C01321 V=800.0 PL=0
MOVL C01322 V=800.0 PL=0
MOVL C01323 V=800.0 PL=0
MOVL C01324 V=800.0 PL=0
MOVL C01325 V=800.0 PL=0
MOVL C01326 V=800.0 PL=0
MOVL C01327 V=800.0 PL=0
MOVL C01328 V=800.0 PL=0
MOVL C01329 V=800.0 PL=0
MOVL C01330 V=800.0 PL=0
MOVL C01331 V=800.0 PL=0
MOVL C01332 V=800.0 PL=0
MOVL C01333 V=800.0 PL=0
MOVL C01334 V=800.0 PL=0
MOVL C01335 V=800.0 PL=0
MOVL C01336 V=800.0 PL=0
MOVL C01337 V=800.0 PL=0
MOVL C01338 V=800.0 PL=0
MOVL C01339 V=800.0 PL=0
MOVL C01340 V=800.0 PL=0
MOVL C01341 V=800.0 PL=0
MOVL C01342 V=800.0 PL=0
MOVL C01343 V=800.0 PL=0
MOVL C01344 V=800.0 PL=0
MOVL C01345 V=800.0 PL=0
MOVL C01346 V=800.0 PL=0
MOVL C01347 V=800.0 PL=0
MOVL C01348 V=800.0 PL=0
MOVL C01349 V=800.0 PL=0
MOVL C01350 V=800.0 PL=0
MOVL C01351 V=800.0 PL=0
MOVL C01352 V=800.0 PL=0
MOVL C01353 V=800.0 PL=0
MOVL C01354 V=800.0 PL=0
MOVL C01355 V=800.0 PL=0
MOVL C01356 V=800.0 PL=0
MOVL C01357 V=800.0 PL=0
MOVL C01358 V=800.0 PL=0
MOVL C01359 V=800.0 PL=0
MOVL C01360 V=800.0 PL=0
MOVL C01361 V=800.0 PL=0
MOVL C01362 V=800.0 PL=0
MOVL C01363 V=800.0 PL=0
MOVL C01364 V=800.0 PL=0
MOVL C01365 V=800.0 PL=0
MOVL C01366 V=800.0 PL=0
MOVL C01367 V=800.0 PL=0
MOVL C01368 V=800.0 PL=0
MOVL C01369 V=800.0 PL=0
MOVL C01370 V=800.0 PL=0
MOVL C01371 V=800.0 PL=0
MOVL C01372 V=800.0 PL=0
MOVL C01373 V=800.0 PL=0
MOVL C01374 V=800.0 PL=0
MOVL C01375 V=800.0 PL=0
MOVL C01376 V=800.0 PL=0
MOVL C01377 V=800.0 PL=0
MOVL C01378 V=800.0 PL=0
MOVL C01379 V=800.0 PL=0
MOVL C01380 V=800.0 PL=0
MOVL C01381 V=800.0 PL=0
MOVL C01382 V=800.0 PL=0
MOVL C01383 V=800.0 PL=0
MOVL C01384 V=800.0 PL=0
MOVL C01385 V=800.0 PL=0
MOVL C01386 V=800.0 PL=0
MOVL C01387 V=800.0 PL=0
MOVL C01388 V=800.0 PL=0
MOVL C01389 V=800.0 PL=0
MOVL C01390 V=800.0 PL=0
MOVL C01391 V=800.0 PL=0
MOVL C01392 V=800.0 PL=0
MOVL C01393 V=800.0 PL=0
MOVL C01394 V=800.0 PL=0
MOVL C01395 V=800.0 PL=0
MOVL C01396 V=800.0 PL=0
MOVL C01397 V=800.0 PL=0
MOVL C01398 V=800.0 PL=0
MOVL C01399 V=800.0 PL=0
MOVL C01400 V=800.0 PL=0
MOVL C01401 V=800.0 PL=0
MOVL C01402 V=800.0 PL=0
MOVL C01403 V=800.0 PL=0
MOVL C01404 V=800.0 PL=0
MOVL C01405 V=800.0 PL=0
MOVL C01406 V=800.0 PL=0
MOVL C01407 V=800.0 PL=0
MOVL C01408 V=800.0 PL=0
MOVL C01409 V=800.0 PL=0
MOVL C01410 V=800.0 PL=0
MOVL C01411 V=800.0 PL=0
MOVL C01412 V=800.0 PL=0
MOVL C01413 V=800.0 PL=0
MOVL C01414 V=800.0 PL=0
MOVL C01415 V=800.0 PL=0
MOVL C01416 V=800.0 PL=0
MOVL C01417 V=800.0 PL=0
MOVL C01418 V=800.0 PL=0
MOVL C01419 V=800.0 PL=0
MOVL C01420 V=800.0 PL=0
MOVL C01421 V=800.0 PL=0
MOVL C01422 V=800.0 PL=0
MOVL C01423 V=800.0 PL=0
MOVL C01424 V=800.0 PL=0
MOVL C01425 V=800.0 PL=0
MOVL C01426 V=800.0 PL=0
MOVL C01427 V=800.0 PL=0
MOVL C01428 V=800.0 PL=0
MOVL C01429 V=800.0 PL=0
MOVL C01430 V=800.0 PL=0
MOVL C01431 V=800.0 PL=0
MOVL C01432 V=800.0 PL=0
MOVL C01433 V=800.0 PL=0
MOVL C01434 V=800.0 PL=0
MOVL C01435 V=800.0 PL=0
MOVL C01436 V=800.0 PL=0
MOVL C01437 V=800.0 PL=0
MOVL C01438 V=800.0 PL=0
MOVL C01439 V=800.0 PL=0
MOVL C01440 V=800.0 PL=0
MOVL C01441 V=800.0 PL=0
MOVL C01442 V=800.0 PL=0
MOVL C01443 V=800.0 PL=0
MOVL C01444 V=800.0 PL=0
MOVL C01445 V=800.0 PL=0
MOVL C01446 V=800.0 PL=0
MOVL C01447 V=800.0 PL=0
MOVL C01448 V=800.0 PL=0
MOVL C01449 V=800.0 PL=0
MOVL C01450 V=800.0 PL=0
MOVL C01451 V=800.0 PL=0
MOVL C01452 V=800.0 PL=0
MOVL C01453 V=800.0 PL=0
MOVL C01454 V=800.0 PL=0
MOVL C01455 V=800.0 PL=0
MOVL C01456 V=800.0 PL=0
MOVL C01457 V=800.0 PL=0
MOVL C01458 V=800.0 PL=0
MOVL C01459 V=800.0 PL=0
MOVL C01460 V=800.0 PL=0
MOVL C01461 V=800.0 PL=0
MOVL C01462 V=800.0 PL=0
MOVL C01463 V=800.0 PL=0
MOVL C01464 V=800.0 PL=0
MOVL C01465 V=800.0 PL=0
MOVL C01466 V=800.0 PL=0
MOVL C01467 V=800.0 PL=0
MOVL C01468 V=800.0 PL=0
MOVL C01469 V=800.0 PL=0
MOVL C01470 V=800.0 PL=0
MOVL C01471 V=800.0 PL=0
MOVL C01472 V=800.0 PL=0
MOVL C01473 V=800.0 PL=0
MOVL C01474 V=800.0 PL=0
MOVL C01475 V=800.0 PL=0
MOVL C01476 V=800.0 PL=0
MOVL C01477 V=800.0 PL=0
MOVL C01478 V=800.0 PL=0
MOVL C01479 V=800.0 PL=0
MOVL C01480 V=800.0 PL=0
MOVL C01481 V=800.0 PL=0
MOVL C01482 V=800.0 PL=0
MOVL C01483 V=800.0 PL=0
MOVL C01484 V=800.0 PL=0
MOVL C01485 V=800.0 PL=0
MOVL C01486 V=800.0 PL=0
MOVL C01487 V=800.0 PL=0
MOVL C01488 V=800.0 PL=0
MOVL C01489 V=800.0 PL=0
MOVL C01490 V=800.0 PL=0
MOVL C01491 V=800.0 PL=0
MOVL C01492 V=800.0 PL=0
MOVL C01493 V=800.0 PL=0
MOVL C01494 V=800.0 PL=0
MOVL C01495 V=800.0 PL=0
MOVL C01496 V=800.0 PL=0
MOVL C01497 V=800.0 PL=0
MOVL C01498 V=800.0 PL=0
MOVL C01499 V=800.0 PL=0
MOVL C01500 V=800.0 PL=0
MOVL C01501 V=800.0 PL=0
MOVL C01502 V=800.0 PL=0
MOVL C01503 V=800.0 PL=0
MOVL C01504 V=800.0 PL=0
MOVL C01505 V=800.0 PL=0
MOVL C01506 V=800.0 PL=0
MOVL C01507 V=800.0 PL=0
MOVL C01508 V=800.0 PL=0
MOVL C01509 V=800.0 PL=0
MOVL C01510 V=800.0 PL=0
MOVL C01511 V=800.0 PL=0
MOVL C01512 V=800.0 PL=0
MOVL C01513 V=800.0 PL=0
MOVL C01514 V=800.0 PL=0
MOVL C01515 V=800.0 PL=0
MOVL C01516 V=800.0 PL=0
MOVL C01517 V=800.0 PL=0
MOVL C01518 V=800.0 PL=0
MOVL C01519 V=800.0 PL=0
MOVL C01520 V=800.0 PL=0
MOVL C01521 V=800.0 PL=0
MOVL C01522 V=800.0 PL=0
MOVL C01523 V=800.0 PL=0
MOVL C01524 V=800.0 PL=0
MOVL C01525 V=800.0 PL=0
MOVL C01526 V=800.0 PL=0
MOVL C01527 V=800.0 PL=0
MOVL C01528 V=800.0 PL=0
MOVL C01529 V=800.0 PL=0
MOVL C01530 V=800.0 PL=0
MOVL C01531 V=800.0 PL=0
MOVL C01532 V=800.0 PL=0
MOVL C01533 V=800.0 PL=0
MOVL C01534 V=800.0 PL=0
MOVL C01535 V=800.0 PL=0
MOVL C01536 V=800.0 PL=0
MOVL C01537 V=800.0 PL=0
MOVL C01538 V=800.0 PL=0
MOVL C01539 V=800.0 PL=0
MOVL C01540 V=800.0 PL=0
MOVL C01541 V=800.0 PL=0
MOVL C01542 V=800.0 PL=0
MOVL C01543 V=800.0 PL=0
MOVL C01544 V=800.0 PL=0
MOVL C01545 V=800.0 PL=0
MOVL C01546 V=800.0 PL=0
MOVL C01547 V=800.0 PL=0
MOVL C01548 V=800.0 PL=0
MOVL C01549 V=800.0 PL=0
MOVL C01550 V=800.0 PL=0
MOVL C01551 V=800.0 PL=0
MOVL C01552 V=800.0 PL=0
MOVL C01553 V=800.0 PL=0
MOVL C01554 V=800.0 PL=0
MOVL C01555 V=800.0 PL=0
MOVL C01556 V=800.0 PL=0
MOVL C01557 V=800.0 PL=0
MOVL C01558 V=800.0 PL=0
MOVL C01559 V=800.0 PL=0
MOVL C01560 V=800.0 PL=0
MOVL C01561 V=800.0 PL=0
MOVL C01562 V=800.0 PL=0
MOVL C01563 V=800.0 PL=0
MOVL C01564 V=800.0 PL=0
MOVL C01565 V=800.0 PL=0
MOVL C01566 V=800.0 PL=0
MOVL C01567 V=800.0 PL=0
MOVL C01568 V=800.0 PL=0
MOVL C01569 V=800.0 PL=0
MOVL C01570 V=800.0 PL=0
MOVL C01571 V=800.0 PL=0
MOVL C01572 V=800.0 PL=0
MOVL C01573 V=800.0 PL=0
MOVL C01574 V=800.0 PL=0
MOVL C01575 V=800.0 PL=0
MOVL C01576 V=800.0 PL=0
MOVL C01577 V=800.0 PL=0
MOVL C01578 V=800.0 PL=0
MOVL C01579 V=800.0 PL=0
MOVL C01580 V=800.0 PL=0
MOVL C01581 V=800.0 PL=0
MOVL C01582 V=800.0 PL=0
MOVL C01583 V=800.0 PL=0
MOVL C01584 V=800.0 PL=0
MOVL C01585 V=800.0 PL=0
MOVL C01586 V=800.0 PL=0
MOVL C01587 V=800.0 PL=0
MOVL C01588 V=800.0 PL=0
MOVL C01589 V=800.0 PL=0
MOVL C01590 V=800.0 PL=0
MOVL C01591 V=800.0 PL=0
MOVL C01592 V=800.0 PL=0
MOVL C01593 V=800.0 PL=0
MOVL C01594 V=800.0 PL=0
MOVL C01595 V=800.0 PL=0
MOVL C01596 V=800.0 PL=0
MOVL C01597 V=800.0 PL=0
MOVL C01598 V=800.0 PL=0
MOVL C01599 V=800.0 PL=0
MOVL C01600 V=800.0 PL=0
MOVL C01601 V=800.0 PL=0
MOVL C01602 V=800.0 PL=0
MOVL C01603 V=800.0 PL=0
MOVL C01604 V=800.0 PL=0
MOVL C01605 V=800.0 PL=0
MOVL C01606 V=800.0 PL=0
MOVL C01607 V=800.0 PL=0
MOVL C01608 V=800.0 PL=0
MOVL C01609 V=800.0 PL=0
MOVL C01610 V=800.0 PL=0
MOVL C01611 V=800.0 PL=0
MOVL C01612 V=800.0 PL=0
MOVL C01613 V=800.0 PL=0
MOVL C01614 V=800.0 PL=0
MOVL C01615 V=800.0 PL=0
MOVL C01616 V=800.0 PL=0
MOVL C01617 V=800.0 PL=0
MOVL C01618 V=800.0 PL=0
MOVL C01619 V=800.0 PL=0
MOVL C01620 V=800.0 PL=0
MOVL C01621 V=800.0 PL=0
MOVL C01622 V=800.0 PL=0
MOVL C01623 V=800.0 PL=0
MOVL C01624 V=800.0 PL=0
MOVL C01625 V=800.0 PL=0
MOVL C01626 V=800.0 PL=0
MOVL C01627 V=800.0 PL=0
MOVL C01628 V=800.0 PL=0
MOVL C01629 V=800.0 PL=0
MOVL C01630 V=800.0 PL=0
MOVL C01631 V=800.0 PL=0
MOVL C01632 V=800.0 PL=0
MOVL C01633 V=800.0 PL=0
MOVL C01634 V=800.0 PL=0
MOVL C01635 V=800.0 PL=0
MOVL C01636 V=800.0 PL=0
MOVL C01637 V=800.0 PL=0
MOVL C01638 V=800.0 PL=0
MOVL C01639 V=800.0 PL=0
MOVL C01640 V=800.0 PL=0
MOVL C01641 V=800.0 PL=0
MOVL C01642 V=800.0 PL=0
MOVL C01643 V=800.0 PL=0
MOVL C01644 V=800.0 PL=0
MOVL C01645 V=800.0 PL=0
MOVL C01646 V=800.0 PL=0
MOVL C01647 V=800.0 PL=0
MOVL C01648 V=800.0 PL=0
MOVL C01649 V=800.0 PL=0
MOVL C01650 V=800.0 PL=0
MOVL C01651 V=800.0 PL=0
MOVL C01652 V=800.0 PL=0
MOVL C01653 V=800.0 PL=0
MOVL C01654 V=800.0 PL=0
MOVL C01655 V=800.0 PL=0
MOVL C01656 V=800.0 PL=0
MOVL C01657 V=800.0 PL=0
MOVL C01658 V=800.0 PL=0
MOVL C01659 V=800.0 PL=0
MOVL C01660 V=800.0 PL=0
MOVL C01661 V=800.0 PL=0
MOVL C01662 V=800.0 PL=0
MOVL C01663 V=800.0 PL=0
MOVL C01664 V=800.0 PL=0
MOVL C01665 V=800.0 PL=0
MOVL C01666 V=800.0 PL=0
MOVL C01667 V=800.0 PL=0
MOVL C01668 V=800.0 PL=0
MOVL C01669 V=800.0 PL=0
MOVL C01670 V=800.0 PL=0
MOVL C01671 V=800.0 PL=0
MOVL C01672 V=800.0 PL=0
MOVL C01673 V=800.0 PL=0
MOVL C01674 V=800.0 PL=0
MOVL C01675 V=800.0 PL=0
MOVL C01676 V=800.0 PL=0
MOVL C01677 V=800.0 PL=0
MOVL C01678 V=800.0 PL=0
MOVL C01679 V=800.0 PL=0
